{attribute 'global_init_slot' := '40510'}
VAR_GLOBAL
  TxTPlant_Facade_sObjectName                                            :T_BA_StateText:='FAS';
  TxTPlant_Facade_sDescription                                            :T_BA_StateText:='Fassade';
  TxTPlant_Natural_smoke_extraction_sObjectName                          :T_BA_StateText:='NRA';
  TxTPlant_Natural_smoke_extraction_sDescription                          :T_BA_StateText:='Natürlicher Rauchabzug';
  TxTPlant_Doors_gates_sluices_sObjectName                               :T_BA_StateText:='TUE';
  TxTPlant_Doors_gates_sluices_sDescription                               :T_BA_StateText:='Türen, Tore, Schleusen';
  TxTPlant_Smoke_and_heat_extraction_system_sObjectName                  :T_BA_StateText:='RWA';
  TxTPlant_Smoke_and_heat_extraction_system_sDescription                  :T_BA_StateText:='Rauch- und Wärmeabzugsanlage';
  TxTPlant_Sunlight_protection_sObjectName                               :T_BA_StateText:='SON';
  TxTPlant_Sunlight_protection_sDescription                               :T_BA_StateText:='Sonnenschutzanlage';
// 411 Abwasseranlagen
  TxTPlant_Separator_facility_sObjectName                                :T_BA_StateText:='ABS';
  TxTPlant_Separator_facility_sDescription                                :T_BA_StateText:='Abscheideranlage';
  TxTPlant_Lifting_system_sObjectName                                    :T_BA_StateText:='HBA';
  TxTPlant_Lifting_system_sDescription                                    :T_BA_StateText:='Hebeanlage';
  TxTPlant_Neutralisation_plant_sObjectName                              :T_BA_StateText:='NEU';
  TxTPlant_Neutralisation_plant_sDescription                              :T_BA_StateText:='Neutralisationsanlage';
// 412 Wasseranlagen
  TxTPlant_Trace_heating_sObjectName                                     :T_BA_StateText:='BGH';
  TxTPlant_Trace_heating_sDescription                                     :T_BA_StateText:='Begleitheizung';
  TxTPlant_Process_water_sObjectName                                     :T_BA_StateText:='BTW';
  TxTPlant_Process_water_sDescription                                     :T_BA_StateText:='Betriebswasser';
  TxTPlant_Well_water_sObjectName                                        :T_BA_StateText:='BWA';
  TxTPlant_Well_water_sDescription                                        :T_BA_StateText:='Brunnenwasser';
  TxTPlant_Dispensing_installation_sObjectName                           :T_BA_StateText:='DOS';
  TxTPlant_Dispensing_installation_sDescription                           :T_BA_StateText:='Dosieranlage';
  TxTPlant_Pressure_booster_system_sObjectName                           :T_BA_StateText:='DEA';
  TxTPlant_Pressure_booster_system_sDescription                           :T_BA_StateText:='Druckerhöhungsanlage';
  TxTPlant_Softening_unit_sObjectName                                    :T_BA_StateText:='EHA';
  TxTPlant_Softening_unit_sDescription                                    :T_BA_StateText:='Enthärtungsanlage';
// Trinkwasser
  TxTPlant_Drinking_water_heating_system_sObjectName                     :T_BA_StateText:='TWE';
  TxTPlant_Drinking_water_heating_system_sDescription                     :T_BA_StateText:='Trinkwassererwärmungsanlage';
  TxTPlant_Reverse_osmosis_system_sObjectName                            :T_BA_StateText:='UKO';
  TxTPlant_Reverse_osmosis_system_sDescription                            :T_BA_StateText:='Umkehrosmoseanlage';
  TxTPlant_Desalination_plant_sObjectName                                :T_BA_StateText:='VEA';
  TxTPlant_Desalination_plant_sDescription                                :T_BA_StateText:='Vollentsalzungsanlage';
// 421 Wärmeerzeugungsanlagen
  TxTPlant_BHKW_sObjectName                                              :T_BA_StateText:='BHK';
  TxTPlant_BHKW_sDescription                                              :T_BA_StateText:='BHKW';
  TxTPlant_Electric_heating_sObjectName                                  :T_BA_StateText:='EHZ';
  TxTPlant_Electric_heating_sDescription                                  :T_BA_StateText:='Elektroheizung';
  TxTPlant_District_heating_transfer_sObjectName                         :T_BA_StateText:='FWÜ';
  TxTPlant_District_heating_transfer_sDescription                         :T_BA_StateText:='Fernwärmeübergabe';
// Geothermieanlage
  TxTPlant_Boiler_sObjectName                                            :T_BA_StateText:='KES';
  TxTPlant_Boiler_sDescription                                            :T_BA_StateText:='Kessel';
  TxTPlant_Clean_steam_generation_sObjectName                            :T_BA_StateText:='RDE';
  TxTPlant_Clean_steam_generation_sDescription                            :T_BA_StateText:='Reindampferzeugung';
  TxTPlant_Solar_power_system_sObjectName                                :T_BA_StateText:='SOL';
  TxTPlant_Solar_power_system_sDescription                                :T_BA_StateText:='Solaranlage';
  TxTPlant_Heating_pump_sObjectName                                      :T_BA_StateText:='WPU';
  TxTPlant_Heating_pump_sDescription                                      :T_BA_StateText:='Wärmepumpe';
// 422 Wärmeverteilnetze
  TxTPlant_Pressure_maintenance_sObjectName                              :T_BA_StateText:='DHG';
  TxTPlant_Pressure_maintenance_sDescription                              :T_BA_StateText:='Druckhaltung';
  TxTPlant_Heating_circuit_sObjectName                                   :T_BA_StateText:='HZK';
  TxTPlant_Heating_circuit_sDescription                                   :T_BA_StateText:='Heizkreis';
  TxTPlant_Heating_sObjectName                                           :T_BA_StateText:='HZG';
  TxTPlant_Heating_sDescription                                           :T_BA_StateText:='Heizung';
  TxTPlant_Back_feed_system_sObjectName                                  :T_BA_StateText:='NSA';
  TxTPlant_Back_feed_system_sDescription                                  :T_BA_StateText:='Nachspeiseanlage';
  TxTPlant_Buffer_sObjectName                                            :T_BA_StateText:='PFS';
  TxTPlant_Buffer_sDescription                                            :T_BA_StateText:='Pufferspeicher';
  TxTPlant_Heat_distribution_network_sObjectName                         :T_BA_StateText:='WVN';
  TxTPlant_Heat_distribution_network_sDescription                         :T_BA_StateText:='Wärmeverteilnetz';
  TxTPlant_Heat_exchanger_sObjectName                                    :T_BA_StateText:='WTR';
  TxTPlant_Heat_exchanger_sDescription                                    :T_BA_StateText:='Wärmeüberträger';
// 423 Raumheizflächen
  TxTPlant_Concrete_core_activation_sObjectName                          :T_BA_StateText:='BKA';
  TxTPlant_Concrete_core_activation_sDescription                          :T_BA_StateText:='Betonkernaktivierung';
  TxTPlant_Overhead_heating_sObjectName                                  :T_BA_StateText:='DHZ';
  TxTPlant_Overhead_heating_sDescription                                  :T_BA_StateText:='Deckenheizung';
  TxTPlant_Ceiling_radiator_panels_sObjectName                           :T_BA_StateText:='DSP';
  TxTPlant_Ceiling_radiator_panels_sDescription                           :T_BA_StateText:='Deckenstrahlplatten';
  TxTPlant_Facade_heating_sObjectName                                    :T_BA_StateText:='FAH';
  TxTPlant_Facade_heating_sDescription                                    :T_BA_StateText:='Fassadenheizung';
  TxTPlant_Panel_heating_sObjectName                                     :T_BA_StateText:='FLH';
  TxTPlant_Panel_heating_sDescription                                     :T_BA_StateText:='Flächenheizung';
  TxTPlant_Underfloor_heating_sObjectName                                :T_BA_StateText:='FBH';
  TxTPlant_Underfloor_heating_sDescription                                :T_BA_StateText:='Fußbodenheizung';
  TxTPlant_Heated_chilled_ceiling_sObjectName                            :T_BA_StateText:='HKD';
  TxTPlant_Heated_chilled_ceiling_sDescription                            :T_BA_StateText:='Heiz-/Kühldecke';
  TxTPlant_Static_heating_sObjectName                                    :T_BA_StateText:='STH';
  TxTPlant_Static_heating_sDescription                                    :T_BA_StateText:='Statische Heizung';
// 430 Lufttechnische Anlagen
  TxTPlant_Extract_air_system_sObjectName                                :T_BA_StateText:='ABA';
  TxTPlant_Extract_air_system_sDescription                                :T_BA_StateText:='Abluftanlage';
  TxTPlant_Roof_air_heater_sObjectName                                   :T_BA_StateText:='DLH';
  TxTPlant_Roof_air_heater_sDescription                                   :T_BA_StateText:='Deckenlufterhitzer';
  TxTPlant_Circulatory_system_sObjectName                                :T_BA_StateText:='KVS';
  TxTPlant_Circulatory_system_sDescription                                :T_BA_StateText:='Kreislaufverbundsystem';
  TxTPlant_Air_processing_unit_sObjectName                               :T_BA_StateText:='LAZ';
  TxTPlant_Air_processing_unit_sDescription                               :T_BA_StateText:='Luftaufbereitungszentrale';
  TxTPlant_Mechanical_smoke_extraction_system_sObjectName                :T_BA_StateText:='MRA';
  TxTPlant_Mechanical_smoke_extraction_system_sDescription                :T_BA_StateText:='Maschinelle Rauchabzugsanlage';
  TxTPlant_Smoke_pressure_system_sObjectName                             :T_BA_StateText:='RDA';
  TxTPlant_Smoke_pressure_system_sDescription                             :T_BA_StateText:='Rauchdruckanlage';
  TxTPlant_Air_handling_unit_sObjectName                                 :T_BA_StateText:='RLT';
  TxTPlant_Air_handling_unit_sDescription                                 :T_BA_StateText:='Raumlufttechnik';
  TxTPlant_Partial_air_conditioning_system_sObjectName                   :T_BA_StateText:='TKA';
  TxTPlant_Partial_air_conditioning_system_sDescription                   :T_BA_StateText:='Teilklimaanlage';
  TxTPlant_Air_curtain_system_sObjectName                                :T_BA_StateText:='TLS';
  TxTPlant_Air_curtain_system_sDescription                                :T_BA_StateText:='Türluftschleieranlage';
  TxTPlant_Recirculating_air_system_sObjectName                          :T_BA_StateText:='ULA';
  TxTPlant_Recirculating_air_system_sDescription                          :T_BA_StateText:='Umluftanlage';
  TxTPlant_Full_air_conditioning_system_sObjectName                      :T_BA_StateText:='VKA';
  TxTPlant_Full_air_conditioning_system_sDescription                      :T_BA_StateText:='Vollklimaanlage';
  TxTPlant_Heat_recovery_system_sObjectName                              :T_BA_StateText:='WRG';
  TxTPlant_Heat_recovery_system_sDescription                              :T_BA_StateText:='Wärmerückgewinnungssystem';
  TxTPlant_Intake_air_system_sObjectName                                 :T_BA_StateText:='ZUA';
  TxTPlant_Intake_air_system_sDescription                                 :T_BA_StateText:='Zuluftanlage';
  TxTPlant_Smoke_extraction_system_sObjectName                           :T_BA_StateText:='ERA';
  TxTPlant_Smoke_extraction_system_sDescription                           :T_BA_StateText:='Entrauchungsanlage';
// 434 Kälteanlagen
  TxTPlant_Remote_cooling_transfer_sObjectName                           :T_BA_StateText:='FKÜ';
  TxTPlant_Remote_cooling_transfer_sDescription                           :T_BA_StateText:='Fernkälteübergabe';
  TxTPlant_Cooling_sObjectName                                           :T_BA_StateText:='KAE';
  TxTPlant_Cooling_sDescription                                           :T_BA_StateText:='Kälte';
  TxTPlant_Cooling_circuit_sObjectName                                   :T_BA_StateText:='KKR';
  TxTPlant_Cooling_circuit_sDescription                                   :T_BA_StateText:='Kältekreis';
  TxTPlant_Cooling_distribution_network_sObjectName                      :T_BA_StateText:='KVN';
  TxTPlant_Cooling_distribution_network_sDescription                      :T_BA_StateText:='Kälteverteilnetz';
  TxTPlant_Cold_water_generation_sObjectName                             :T_BA_StateText:='KWE';
  TxTPlant_Cold_water_generation_sDescription                             :T_BA_StateText:='Kaltwassererzeugung';
  TxTPlant_Electrical_cabinet_cooling_sObjectName                        :T_BA_StateText:='KVE';
  TxTPlant_Electrical_cabinet_cooling_sDescription                        :T_BA_StateText:='Kühlung Schaltschrank ';
  TxTPlant_Cooling_storage_sObjectName                                   :T_BA_StateText:='KSP';
  TxTPlant_Cooling_storage_sDescription                                   :T_BA_StateText:='Kältespeicher';
  TxTPlant_Chilled_ceiling_sObjectName                                   :T_BA_StateText:='KÜD';
  TxTPlant_Chilled_ceiling_sDescription                                   :T_BA_StateText:='Kühldecke';
  TxTPlant_Re_cooling_plant_sObjectName                                  :T_BA_StateText:='RKW';
  TxTPlant_Re_cooling_plant_sDescription                                  :T_BA_StateText:='Rückkühlwerk';
// 441 Hoch- und Mittelspannungsanlagen
  TxTPlant_Switchgear_sObjectName                                        :T_BA_StateText:='STA';
  TxTPlant_Switchgear_sDescription                                        :T_BA_StateText:='Schaltanlagen';
  TxTPlant_Transformer_sObjectName                                       :T_BA_StateText:='TRF';
  TxTPlant_Transformer_sDescription                                       :T_BA_StateText:='Transformator';
  TxTPlant_Medium_voltage_system_sObjectName                             :T_BA_StateText:='MSA';
  TxTPlant_Medium_voltage_system_sDescription                             :T_BA_StateText:='Mittelspannungsanlage';
  TxTPlant_Compensation_system_sObjectName                               :T_BA_StateText:='KOA';
  TxTPlant_Compensation_system_sDescription                               :T_BA_StateText:='Kompensationsanlage';
  TxTPlant_Frequency_converter_system_sObjectName                        :T_BA_StateText:='FUA';
  TxTPlant_Frequency_converter_system_sDescription                        :T_BA_StateText:='Frequenzumformeranlage';
// 442 Eigenstromversorgungsanlagen
  TxTPlant_Emissions_system_sObjectName                                  :T_BA_StateText:='AGA';
  TxTPlant_Emissions_system_sDescription                                  :T_BA_StateText:='Abgasanlage';
  TxTPlant_Battery_unit_sObjectName                                      :T_BA_StateText:='BAT';
  TxTPlant_Battery_unit_sDescription                                      :T_BA_StateText:='Batterieanlage';
  TxTPlant_Co_generation_unit_sObjectName                                :T_BA_StateText:='BHK';
  TxTPlant_Co_generation_unit_sDescription                                :T_BA_StateText:='Blockheizkraftwerk';
  TxTPlant_Fuel_supply_sObjectName                                       :T_BA_StateText:='BRV';
  TxTPlant_Fuel_supply_sDescription                                       :T_BA_StateText:='Brennstoffversorgung';
  TxTPlant_Standby_power_system_sObjectName                              :T_BA_StateText:='ESA';
  TxTPlant_Standby_power_system_sDescription                              :T_BA_StateText:='Ersatzstromanlage';
  TxTPlant_Photovoltaic_system_sObjectName                               :T_BA_StateText:='PVA';
  TxTPlant_Photovoltaic_system_sDescription                               :T_BA_StateText:='Fotovoltaikanlage';
  TxTPlant_Uninterruptible_power_supply_sObjectName                      :T_BA_StateText:='USV';
  TxTPlant_Uninterruptible_power_supply_sDescription                      :T_BA_StateText:='Unterbrechungsfreie Stromversorgung';
// 443 Niederspannungsschaltanlagen
  TxTPlant_General_power_supply_sObjectName                              :T_BA_StateText:='ASV';
  TxTPlant_General_power_supply_sDescription                              :T_BA_StateText:='Allgemeine Stromversorgung';
  TxTPlant_Safety_power_supply_sObjectName                               :T_BA_StateText:='SSV';
  TxTPlant_Safety_power_supply_sDescription                               :T_BA_StateText:='Sicherheitsstromversorgung';
  TxTPlant_Lighting_sObjectName                                          :T_BA_StateText:='BEL';
  TxTPlant_Lighting_sDescription                                          :T_BA_StateText:='Beleuchtungsanlage';
  TxTPlant_Emergency_lighting_sObjectName                                :T_BA_StateText:='SIB';
  TxTPlant_Emergency_lighting_sDescription                                :T_BA_StateText:='Sicherheitsbeleuchtung';
// 451 Telekommunikationsanlagen
  TxTPlant_Telecommunications_system_sObjectName                         :T_BA_StateText:='TEL';
  TxTPlant_Telecommunications_system_sDescription                         :T_BA_StateText:='Telekommunikationsanlage';
// 452 Such- und Signalanlagen
  TxTPlant_Call_signalling_system_sObjectName                            :T_BA_StateText:='LRA';
  TxTPlant_Call_signalling_system_sDescription                            :T_BA_StateText:='Lichtrufanlage';
  TxTPlant_Door_intercom_and_door_opener_system_sObjectName              :T_BA_StateText:='TÜA';
  TxTPlant_Door_intercom_and_door_opener_system_sDescription              :T_BA_StateText:='Türsprech- und -öffneranlage';
  TxTPlant_Paging_system_sObjectName                                     :T_BA_StateText:='PRA';
  TxTPlant_Paging_system_sDescription                                     :T_BA_StateText:='Personenrufanlage';
// 453 Zeitdienstanlagen
  TxTPlant_Clock_and_time_recording_system_sObjectName                   :T_BA_StateText:='ZEA';
  TxTPlant_Clock_and_time_recording_system_sDescription                   :T_BA_StateText:='Uhren- und Zeiterfassungsanlage';
// 454 Elektroakustische Anlagen
  TxTPlant_Electro_acoustic_sound_systems_sObjectName                    :T_BA_StateText:='ELA';
  TxTPlant_Electro_acoustic_sound_systems_sDescription                    :T_BA_StateText:='Elektroakustische Anl. , Beschallung';
  TxTPlant_Conference_and_interpreting_equipment_sObjectName             :T_BA_StateText:='KDA';
  TxTPlant_Conference_and_interpreting_equipment_sDescription             :T_BA_StateText:='Konferenz- und Dolmetscheranlage';
  TxTPlant_Intercom_system_sObjectName                                   :T_BA_StateText:='GSA';
  TxTPlant_Intercom_system_sDescription                                   :T_BA_StateText:='Gegensprechanlage';
  TxTPlant_Voice_alarm_system_sObjectName                                :T_BA_StateText:='SAA';
  TxTPlant_Voice_alarm_system_sDescription                                :T_BA_StateText:='Sprachalarmierungsanlage';
  TxTPlant_Intercommunication_systems_sObjectName                        :T_BA_StateText:='WSA';
  TxTPlant_Intercommunication_systems_sDescription                        :T_BA_StateText:='Wechselsprechanlagen';
// 455 Fernseh- und Antennenanlagen
  TxTPlant_Television_system_sObjectName                                 :T_BA_StateText:='TVA';
  TxTPlant_Television_system_sDescription                                 :T_BA_StateText:='Fernsehanlage';
  TxTPlant_Transmitting_and_receiving_antenna_system_sObjectName         :T_BA_StateText:='SEA';
  TxTPlant_Transmitting_and_receiving_antenna_system_sDescription         :T_BA_StateText:='Sende- und Empfangsantennenanlage';
  TxTPlant_BOS_radio_system_sObjectName                                  :T_BA_StateText:='BOS';
  TxTPlant_BOS_radio_system_sDescription                                  :T_BA_StateText:='BOS-Funkanlage';
// 456 Gefahrenmelde- und Alarmanlagen
  TxTPlant_Fire_detection_and_alarm_system_sObjectName                   :T_BA_StateText:='BMA';
  TxTPlant_Fire_detection_and_alarm_system_sDescription                   :T_BA_StateText:='Brandmeldeanlage';
  TxTPlant_Carbon_monoxide_warning_system_sObjectName                    :T_BA_StateText:='COW';
  TxTPlant_Carbon_monoxide_warning_system_sDescription                    :T_BA_StateText:='CO-Warnanlage';
  TxTPlant_Burglar_alarm_system_sObjectName                              :T_BA_StateText:='EMA';
  TxTPlant_Burglar_alarm_system_sDescription                              :T_BA_StateText:='Einbruchmeldeanlage';
  TxTPlant_Fire_control_panel_sObjectName                                :T_BA_StateText:='FWT';
  TxTPlant_Fire_control_panel_sDescription                                :T_BA_StateText:='Feuerwehrtableau';
  TxTPlant_Escape_route_protection_system_sObjectName                    :T_BA_StateText:='FWS';
  TxTPlant_Escape_route_protection_system_sDescription                    :T_BA_StateText:='Fluchtwegsicherungsanlage';
  TxTPlant_Hazard_detection_system_sObjectName                           :T_BA_StateText:='GMA';
  TxTPlant_Hazard_detection_system_sDescription                           :T_BA_StateText:='Gefahrenmeldeanlage';
  TxTPlant_Gas_warning_system_sObjectName                                :T_BA_StateText:='GWA';
  TxTPlant_Gas_warning_system_sDescription                                :T_BA_StateText:='Gaswarnanlage';
  TxTPlant_Smoke_aspiration_system_sObjectName                           :T_BA_StateText:='RAS';
  TxTPlant_Smoke_aspiration_system_sDescription                           :T_BA_StateText:='Rauchansaugsystem';
  TxTPlant_Room_observation_system_sObjectName                           :T_BA_StateText:='RBA';
  TxTPlant_Room_observation_system_sDescription                           :T_BA_StateText:='Raumbeobachtungsanlage';
  TxTPlant_Robbery_alarm_system_sObjectName                              :T_BA_StateText:='ÜFA';
  TxTPlant_Robbery_alarm_system_sDescription                              :T_BA_StateText:='Überfallmeldeanlage';
  TxTPlant_Guard_control_system_sObjectName                              :T_BA_StateText:='WKA';
  TxTPlant_Guard_control_system_sDescription                              :T_BA_StateText:='Wächterkontrollanlage';
  TxTPlant_Emergency_call_system_sObjectName                             :T_BA_StateText:='NOT';
  TxTPlant_Emergency_call_system_sDescription                             :T_BA_StateText:='Notrufanlage';
  TxTPlant_Access_control_system_sObjectName                             :T_BA_StateText:='ZKS';
  TxTPlant_Access_control_system_sDescription                             :T_BA_StateText:='Zugangskontrollsystem';
// 457 Übertragungsnetze
  TxTPlant_Networks_for_the_transmission_voice_text_etc_sObjectName      :T_BA_StateText:='LAN';
  TxTPlant_Networks_for_the_transmission_voice_text_etc_sDescription      :T_BA_StateText:='Netzw.  Daten, Sprache, Text etc';
// 459 Fernmelde- und informationstechnische Anlagen, Sonstiges
  TxTPlant_Remote_control_systems_sObjectName                            :T_BA_StateText:='FWA';
  TxTPlant_Remote_control_systems_sDescription                            :T_BA_StateText:='Fernwirkanlagen';
  TxTPlant_Parking_guidance_systems_sObjectName                          :T_BA_StateText:='PLS';
  TxTPlant_Parking_guidance_systems_sDescription                          :T_BA_StateText:='Parkleitsysteme';
// 460 Förderanlagen
  TxTPlant_File_transportation_systems_sObjectName                       :T_BA_StateText:='ATA';
  TxTPlant_File_transportation_systems_sDescription                       :T_BA_StateText:='Aktentransportanlagen';
  TxTPlant_Lift_sObjectName                                              :T_BA_StateText:='AUF';
  TxTPlant_Lift_sDescription                                              :T_BA_StateText:='Aufzug';
  TxTPlant_Inspection_systems_sObjectName                                :T_BA_StateText:='BFA';
  TxTPlant_Inspection_systems_sDescription                                :T_BA_StateText:='Befahranlagen';
  TxTPlant_Moving_walkways_sObjectName                                   :T_BA_StateText:='FST';
  TxTPlant_Moving_walkways_sDescription                                   :T_BA_StateText:='Fahrsteige';
  TxTPlant_Escalators_sObjectName                                        :T_BA_StateText:='FTR';
  TxTPlant_Escalators_sDescription                                        :T_BA_StateText:='Fahrtreppen';
  TxTPlant_External_lifts_sObjectName                                    :T_BA_StateText:='FSA';
  TxTPlant_External_lifts_sDescription                                    :T_BA_StateText:='Fassadenaufzüge';
  TxTPlant_Baggage_conveyor_system_sObjectName                           :T_BA_StateText:='GFA';
  TxTPlant_Baggage_conveyor_system_sDescription                           :T_BA_StateText:='Gepäckförderanlage';
  TxTPlant_Pneumatic_delivery_systems_sObjectName                        :T_BA_StateText:='RPA';
  TxTPlant_Pneumatic_delivery_systems_sDescription                        :T_BA_StateText:='Rohrpostanlagen';
  TxTPlant_Goods_transportation_facilities_sObjectName                   :T_BA_StateText:='WTA';
  TxTPlant_Goods_transportation_facilities_sDescription                   :T_BA_StateText:='Warentransportanlagen';
// 470 Nutzerspezifische Anlagen
// 471 Küchentechnische Anlagen
  TxTPlant_Small_refrigeration_unit_sObjectName                          :T_BA_StateText:='KLK';
  TxTPlant_Small_refrigeration_unit_sDescription                          :T_BA_StateText:='Kleinkälteanlage';
// 472 Wäscherei- und Reinigungsanlagen
  TxTPlant_Disinfection_unit_sObjectName                                 :T_BA_StateText:='DES';
  TxTPlant_Disinfection_unit_sDescription                                 :T_BA_StateText:='Desinfektionsanlage';
  TxTPlant_Cleaning_unit_sObjectName                                     :T_BA_StateText:='REA';
  TxTPlant_Cleaning_unit_sDescription                                     :T_BA_StateText:='Reinigungsanlage';
  TxTPlant_Sterilisation_systems_sObjectName                             :T_BA_StateText:='STR';
  TxTPlant_Sterilisation_systems_sDescription                             :T_BA_StateText:='Sterilisationseinrichtungen';
  TxTPlant_Water_treatment_system_sObjectName                            :T_BA_StateText:='WAA';
  TxTPlant_Water_treatment_system_sDescription                            :T_BA_StateText:='Wasseraufbereitungsanlage';
  TxTPlant_Laundry_system_sObjectName                                    :T_BA_StateText:='WÄA';
  TxTPlant_Laundry_system_sDescription                                    :T_BA_StateText:='Wäschereianlage';
// 473 Medienversorgungsanlagen
  TxTPlant_Compressed_air_supply_system_sObjectName                      :T_BA_StateText:='DRL';
  TxTPlant_Compressed_air_supply_system_sDescription                      :T_BA_StateText:='Druckluftversorgungsanlage';
  TxTPlant_Pressure_regulator_unit_sObjectName                           :T_BA_StateText:='DRA';
  TxTPlant_Pressure_regulator_unit_sDescription                           :T_BA_StateText:='Druckregelanlage';
  TxTPlant_Media_supply_system_sObjectName                               :T_BA_StateText:='MVA';
  TxTPlant_Media_supply_system_sDescription                               :T_BA_StateText:='Medienversorgungsanlage';
  TxTPlant_Medical_and_technical_gases_sObjectName                       :T_BA_StateText:='MTG';
  TxTPlant_Medical_and_technical_gases_sDescription                       :T_BA_StateText:='Medizinische und technische Gase';
  TxTPlant_Vacuum_unit_sObjectName                                       :T_BA_StateText:='VAK';
  TxTPlant_Vacuum_unit_sDescription                                       :T_BA_StateText:='Vakuumanlage';
// 474 Medizin- und labortechnische Anlagen
  TxTPlant_Medical_technical_plant_sObjectName                           :T_BA_StateText:='MED';
  TxTPlant_Medical_technical_plant_sDescription                           :T_BA_StateText:='Medizintechnische Anlagen';
  TxTPlant_Medical_gas_supply_sObjectName                                :T_BA_StateText:='MGV';
  TxTPlant_Medical_gas_supply_sDescription                                :T_BA_StateText:='Medizinische Gasversorgung';
  TxTPlant_Laboratory_equipment_sObjectName                              :T_BA_StateText:='LAB';
  TxTPlant_Laboratory_equipment_sDescription                              :T_BA_StateText:='Labortechnische Anlagen (allgemein)';
// 475 Feuerlöschanlagen
  TxTPlant_Fire_extinguisher_sObjectName                                 :T_BA_StateText:='FLA';
  TxTPlant_Fire_extinguisher_sDescription                                 :T_BA_StateText:='Feuerlöschanlage';
  TxTPlant_Gas_extinguishing_system_sObjectName                          :T_BA_StateText:='GLA';
  TxTPlant_Gas_extinguishing_system_sDescription                          :T_BA_StateText:='Gaslöschanlage';
  TxTPlant_Fire_extinguishing_system_sObjectName                         :T_BA_StateText:='LÖS';
  TxTPlant_Fire_extinguishing_system_sDescription                         :T_BA_StateText:='Löschanlage (allgemein)';
  TxTPlant_Mist_extinguishing_system_sObjectName                         :T_BA_StateText:='NLA';
  TxTPlant_Mist_extinguishing_system_sDescription                         :T_BA_StateText:='Nebellöschanlage';
  TxTPlant_NOX_system_sObjectName                                        :T_BA_StateText:='NOX';
  TxTPlant_NOX_system_sDescription                                        :T_BA_StateText:='NOX-Anlage';
  TxTPlant_Sprinkler_system_sObjectName                                  :T_BA_StateText:='SPR';
  TxTPlant_Sprinkler_system_sDescription                                  :T_BA_StateText:='Sprinkleranlage';
  TxTPlant_Wall_hydrant_system_sObjectName                               :T_BA_StateText:='WHA';
  TxTPlant_Wall_hydrant_system_sDescription                               :T_BA_StateText:='Wandhydrantenanlage';
// 478 Entsorgungsanlagen
  TxTPlant_Waste_disposal_system_sObjectName                             :T_BA_StateText:='AEA';
  TxTPlant_Waste_disposal_system_sDescription                             :T_BA_StateText:='Abfallentsorgungsanlage';
  TxTPlant_Media_disposal_system_sObjectName                             :T_BA_StateText:='MEA';
  TxTPlant_Media_disposal_system_sDescription                             :T_BA_StateText:='Medienentsorgungsanlage';
  TxTPlant_Vacuum_cleaning_systems_sObjectName                           :T_BA_StateText:='SSA';
  TxTPlant_Vacuum_cleaning_systems_sDescription                           :T_BA_StateText:='Staubsauganlagen';
// 480 Gebäudeautomation
  TxTPlant_Information_focal_point_sObjectName                           :T_BA_StateText:='ISP';
  TxTPlant_Information_focal_point_sDescription                           :T_BA_StateText:='Informationsschwerpunkt';
  TxTPlant_Weather_station_sObjectName                                   :T_BA_StateText:='WET';
  TxTPlant_Weather_station_sDescription                                   :T_BA_StateText:='Wetterstation';
  TxTPlant_Management_and_operating_equipment_sObjectName                :T_BA_StateText:='MBE';
  TxTPlant_Management_and_operating_equipment_sDescription                :T_BA_StateText:='Management- und Bedieneinrichtungen';
  TxTPlant_Room_automation_sObjectName                                   :T_BA_StateText:='RAU';
  TxTPlant_Room_automation_sDescription                                   :T_BA_StateText:='Raumautomation';
  TxTPlant_Room_automation_system_distributor_sObjectName                :T_BA_StateText:='RAV';
  TxTPlant_Room_automation_system_distributor_sDescription                :T_BA_StateText:='Raumautomation-Systemverteiler';
  TxTPlant_Control_cabinet_sObjectName                                   :T_BA_StateText:='SSK';
  TxTPlant_Control_cabinet_sDescription                                   :T_BA_StateText:='Schaltschrank';
  TxTPlant_Settings_sObjectName                                          :T_BA_StateText:='ALP';
  TxTPlant_Settings_sDescription                                          :T_BA_StateText:='Anlagenparameter';
  TxTPlant_EventGroups_sObjectName                                       :T_BA_StateText:='ERG';
  TxTPlant_EventGroups_sDescription                                       :T_BA_StateText:='Meldeklassen';
  TxTPlant_Global_Building_Data_sObjectName                              :T_BA_StateText:='GGL';
  TxTPlant_Global_Building_Data_sDescription                              :T_BA_StateText:='globale Gebäudedaten';
// 540 Technische Anlagen in Außenanlagen
  TxTPlant_Rainwater_retention_basin_sObjectName                         :T_BA_StateText:='RRB';
  TxTPlant_Rainwater_retention_basin_sDescription                         :T_BA_StateText:='Regenrückhaltebecken';
  TxTPlant_Cistern_system_sObjectName                                    :T_BA_StateText:='ZTA';
  TxTPlant_Cistern_system_sDescription                                    :T_BA_StateText:='Zisternenanlage';
END_VAR

// ---- Templates/GVLs/Language/German/TxtTrade_DE.TcGVL
{region '#Template'}
	{attribute 'Version' := '1.2.0.0'}
	{attribute 'Tags' := '"LCID": "1031", "Text": "GVL, DPAD, Trades, ObjectName, Description"'}
	{attribute 'Tags' := '"LCID": "1033", "Text": "GVL, DPAD, Trades, ObjectName, Description"'}
	{attribute 'Description' := '"LCID": "1031", "Text": "Textliste Gewerke"'}
	{attribute 'Description' := '"LCID": "1033", "Text": "Text list trades"'}
{endregion}

{attribute 'global_init_slot' := '40510'}
VAR_GLOBAL
  TxtTrade_Doors_gates_windows_sun_protection_sObjectName                :T_BA_StateText:='TTF';
  TxtTrade_Doors_gates_windows_sun_protection_sDescription                :T_BA_StateText:='Türen, Tore, Fenster, Sonnenschutz';
  TxtTrade_Sewage_water_and_gas_plants_sObjectName                       :T_BA_StateText:='GWA';
  TxtTrade_Sewage_water_and_gas_plants_sDescription                       :T_BA_StateText:='Abwasser-, Wasser-, Gasanlagen';
  TxtTrade_Heat_supply_systems_sObjectName                               :T_BA_StateText:='HZG';
  TxtTrade_Heat_supply_systems_sDescription                               :T_BA_StateText:='Wärmeversorgungsanlagen';
  TxtTrade_Air_conditioning_sObjectName                                  :T_BA_StateText:='LTA';
  TxtTrade_Air_conditioning_sDescription                                  :T_BA_StateText:='Lufttechnische Anlagen';
  TxtTrade_Refrigeration_systems_sObjectName                             :T_BA_StateText:='KAE';
  TxtTrade_Refrigeration_systems_sDescription                             :T_BA_StateText:='Kälteanlagen';
  TxtTrade_High_voltage_systems_sObjectName                              :T_BA_StateText:='ELT';
  TxtTrade_High_voltage_systems_sDescription                              :T_BA_StateText:='Starkstromanlagen';
  TxtTrade_Telecommunication_and_information_technology_sObjectName      :T_BA_StateText:='FIA';
  TxtTrade_Telecommunication_and_information_technology_sDescription      :T_BA_StateText:='Fernm.- und informationstech. Anlagen';
  TxtTrade_Hazard_detection_and_alarm_systems_sObjectName                :T_BA_StateText:='GMA';
  TxtTrade_Hazard_detection_and_alarm_systems_sDescription                :T_BA_StateText:='Gefahrenmelde- und Alarmanlagen';
  TxtTrade_Conveyors_sObjectName                                         :T_BA_StateText:='FTA';
  TxtTrade_Conveyors_sDescription                                         :T_BA_StateText:='Förderanlagen';
  TxtTrade_Kitchen_technology_systems_sObjectName                        :T_BA_StateText:='KTA';
  TxtTrade_Kitchen_technology_systems_sDescription                        :T_BA_StateText:='Küchentechnische Anlagen';
  TxtTrade_Laundry_and_cleaning_systems_sObjectName                      :T_BA_StateText:='WAR';
  TxtTrade_Laundry_and_cleaning_systems_sDescription                      :T_BA_StateText:='Wäscherei- und Reinigungsanlagen';
  TxtTrade_Media_supply_systems_sObjectName                              :T_BA_StateText:='MVA';
  TxtTrade_Media_supply_systems_sDescription                              :T_BA_StateText:='Medienversorgungsanlagen';
  TxtTrade_Medical_and_laboratory_equipment_sObjectName                  :T_BA_StateText:='MED';
  TxtTrade_Medical_and_laboratory_equipment_sDescription                  :T_BA_StateText:='Medizin- und labortechnische Anlagen';
  TxtTrade_Fire_extinguishing_systems_sObjectName                        :T_BA_StateText:='FLA';
  TxtTrade_Fire_extinguishing_systems_sDescription                        :T_BA_StateText:='Feuerlöschanlagen';
  TxtTrade_Bathing_facilities_sObjectName                                :T_BA_StateText:='BTA';
  TxtTrade_Bathing_facilities_sDescription                                :T_BA_StateText:='Badetechnische Anlagen';
  TxtTrade_Process_heating_cooling_and_air_systems_sObjectName           :T_BA_StateText:='PRO';
  TxtTrade_Process_heating_cooling_and_air_systems_sDescription           :T_BA_StateText:='Prozesswärme-, -kälte- und -luftanlagen';
  TxtTrade_Waste_disposal_facilities_sObjectName                         :T_BA_StateText:='ENT';
  TxtTrade_Waste_disposal_facilities_sDescription                         :T_BA_StateText:='Entsorgungsanlagen';
  TxtTrade_Building_automation_and_control_systems_general_sObjectName   :T_BA_StateText:='GAS';
  TxtTrade_Building_automation_and_control_systems_general_sDescription   :T_BA_StateText:='Gebäudeautomation allgemein';
  TxtTrade_Automation_focal_point_information_focal_point_sObjectName    :T_BA_StateText:='ASP';
  TxtTrade_Automation_focal_point_information_focal_point_sDescription    :T_BA_StateText:='Automationsschwerpunkt';
  TxtTrade_Room_automation_sObjectName                                   :T_BA_StateText:='RAU';
  TxtTrade_Room_automation_sDescription                                   :T_BA_StateText:='Raumautomation';
  TxtTrade_Outdoor_devices_sObjectName                                   :T_BA_StateText:='AUG';
  TxtTrade_Outdoor_devices_sDescription                                   :T_BA_StateText:='Außengeräte';
END_VAR

// ---- Templates/GVLs/Site/Site.TcGVL
{region '#Template'}
	{attribute 'Version' := '1.0.0.0'}
	{attribute 'Tags' := '"LCID": "1031", "Text": "GVL, Publisher, Subscriber"'}
	{attribute 'Tags' := '"LCID": "1033", "Text": "GVL, Publisher, Subscriber"'}
	{attribute 'Description' := '"LCID": "1031", "Text": "Ams NetId, Subject"'}
	{attribute 'Description' := '"LCID": "1033", "Text": "Ams NetId, Subject"'}
{endregion}

{attribute 'qualified_only'}
VAR_GLOBAL	
	Self_NetId						: T_BA_MedString	:= '127.0.0.1.1.1';
	Ipc1_NetId						: T_BA_MedString	:= Self_NetId;
	Ipc2_NetId						: T_BA_MedString	:= Self_NetId;
	Ipc3_NetId						: T_BA_MedString	:= Self_NetId;
	Ipc4_NetId						: T_BA_MedString	:= Self_NetId;
	Ipc5_NetId						: T_BA_MedString	:= Self_NetId;
	                            	
	GeneralSettings_Subject			: T_BA_MedString	:= 'GeneralSettings';	
	GeneralSettings_NetId			: T_BA_MedString	:= Self_NetId;	
		                        	
	WeatherStation_Subject			: T_BA_MedString	:= 'WeatherStation';
	WeatherStation_NetId			: T_BA_MedString	:= Self_NetId;
                                	
	FacadeNorth_NetId				: T_BA_MedString	:= Ipc1_NetId;
	FacadeNorth_Subject				: T_BA_MedString	:= 'FcdNorth.FacadeSunBlind';
	FacadeEast_NetId				: T_BA_MedString	:= Ipc1_NetId;
	FacadeEast_Subject				: T_BA_MedString	:= 'FcdEast.FacadeSunBlind';
	FacadeSouth_NetId				: T_BA_MedString	:= Ipc1_NetId;
	FacadeSouth_Subject				: T_BA_MedString	:= 'FcdSouth.FacadeSunBlind';
	FacadeWest_NetId				: T_BA_MedString	:= Ipc1_NetId;
	FacadeWest_Subject				: T_BA_MedString	:= 'FcdWest.FacadeSunBlind';
                                	
	Building_NetId					: T_BA_MedString	:= Ipc1_NetId;
	BuildingAlarms_Subject			: T_BA_MedString	:= 'BuildingAlarms';
	BuildingMode_Subject			: T_BA_MedString	:= 'BuildingMode';
	BuildingEnergyLevel_Subject		: T_BA_MedString	:= 'BuildingEnergyLevel';
	BuildingSpRmT_Subject			: T_BA_MedString	:= 'BuildingSpRmT';
	BuildingSunProtection_Subject	: T_BA_MedString	:= 'BuildingSunProtection';
END_VAR

// ---- POUs/MAIN.TcPOU
PROGRAM MAIN
VAR
	DPAD		: FB_BA_CarelessDPAD := (
					aIdentifier := [
	(* Level 1 *)		(eMode:=E_BA_DPADMode.eInclude,		eNodeType:=E_BA_NodeType.eLocation,			sSeparator_ObjectName := '-', 	sSeparator_Description := ' - ',	nIndexDigits := 0),
	(* Level 2 *)		(eMode:=E_BA_DPADMode.eInclude,		eNodeType:=E_BA_NodeType.eBuilding,			sSeparator_ObjectName := '-', 	sSeparator_Description := ' - ',	nIndexDigits := 0),
	(* Level 3 *)		(eMode:=E_BA_DPADMode.eInclude,		eNodeType:=E_BA_NodeType.eControlCabinet,	sSeparator_ObjectName := '-', 	sSeparator_Description := ' - ',	nIndexDigits := 0),
	(* Level 4 *)		(eMode:=E_BA_DPADMode.eInclude,		eNodeType:=E_BA_NodeType.eFloor,			sSeparator_ObjectName := '-', 	sSeparator_Description := ' - ',	nIndexDigits := 0),
	(* Level 5 *)		(eMode:=E_BA_DPADMode.eInclude,		eNodeType:=E_BA_NodeType.eTrade,			sSeparator_ObjectName := '-', 	sSeparator_Description := ' - ',	nIndexDigits := 0),
	(* Level 6 *)		(eMode:=E_BA_DPADMode.eInclude,		eNodeType:=E_BA_NodeType.ePlant,			sSeparator_ObjectName := '-', 	sSeparator_Description := ' - ',	nIndexDigits := 0),
	(* Level 7 *)		(eMode:=E_BA_DPADMode.eInclude,		eNodeType:=E_BA_NodeType.eAggregate,		sSeparator_ObjectName := '-', 	sSeparator_Description := ' - ',	nIndexDigits := 2),
	(* Level 8 *)		(eMode:=E_BA_DPADMode.eInclude,		eNodeType:=E_BA_NodeType.eFunction,			sSeparator_ObjectName := '-', 	sSeparator_Description := ' - ',	nIndexDigits := 2)
					]
				);		
		 
//	Level 1 Standort bzw. Ort oder Stadt 
//	Level 1 Site respectively location or town
	SiteA		: FB_BA_View := (
					sObjectName		:= 'A',		
					sDescription	:= 'A',	
					eDPADMode		:= E_BA_DPADMode.eInclude				
				); 				
//	Level 2 Gebäude 	
//	Level 2 Building 	
		B			: FB_BA_View := (
						iParent 		:= SiteA,
						sObjectName		:= 'B',		
						sDescription	:= 'B',	
						eDPADMode		:= E_BA_DPADMode.eInclude					
					);     
// Level 3 ISP -> Informationsschwerpunkt
// Level 3 IFP -> information focal point 	 	                                                                                   	
			IFP			: FB_BA_View := (
							iParent 		:= B,
							sObjectName		:= 'I',		
							sDescription	:= 'IFP',	
							eDPADMode		:= E_BA_DPADMode.eInclude				
						);     
// Level 4 Stockwerk 	->	O01 = Obergeschoss 01, U01 = Untergeschoss 01,  E00 = Ergeschoss
// Level 4 floor ->	F01 = floor 01, B01 = basement 01,  GFL = Ground floor  						
				F01			: FB_BA_View := (
								iParent 		:= IFP,
								sObjectName		:= 'F01',		
								sDescription	:= 'Floor 01',
								eDPADMode		:= E_BA_DPADMode.eInclude					
							);     	
// Level 5 Gewerk Wärmeversorgungsanlagen  
// Level 5 Trade Heat supply systems, heat distribution  --> 	HD = heat distribution, HG = heat generation
					H			: FB_BA_H := (
									iParent 		:= F01,
									sObjectName		:= 'HTG',		
									sDescription	:= 'Heat supply systems',
									eDPADMode		:= E_BA_DPADMode.eInclude			
								);     	 	
// Level 5 Gewerk Gebäudeautomation Allgemein   
// Level 5 Trade General                                                                                       	
					G			: FB_BA_General := (
									iParent 		:= F01,
									sObjectName		:= 'BAG',
									sDescription	:= 'General',
									eDPADMode		:= E_BA_DPADMode.eInclude					
								);     	 											   	 											
// Level 5 Gewerk Luftechnische Anlagen      
// Level 5 Trade ventilation system                                                                                	
					AC			: FB_BA_AC := (
									iParent 		:= F01,
									sObjectName		:= 'AC_',
									sDescription	:= 'Air conditioning',
									eDPADMode		:= E_BA_DPADMode.eInclude
								);     	
// Level 5 Gewerk Raumautomation    
// Level 5 Trade room automation                                                                              	

								
// Level 5 Gewerk Außengeräte   
// Level 5 Trade Outdoor devices     
					OD			: FB_BA_OD := (
									iParent			:= F01,
									sObjectName		:= 'ODD',
									sDescription	:= 'Outdoor devices',
									eDPADMode		:= E_BA_DPADMode.eInclude
								);
END_VAR

//	Level 1 Standort bzw. Ort oder Stadt 	Site respectively location or town
SiteA();
//	Level 2 Gebäude 	Building		
	B();
// Level 3 ISP -> Informationsschwerpunkt	information focal point 
		IFP();
// Level 4 Stockwerk -->	O01 = Obergeschoss 01, U01 = Untergeschoss 01,  E00 = Ergeschoss 	floor ->	F01 = floor 01, B01 = basement 01,  GFL = Ground floor
			F01();
// Level 5 Gewerk Wärmeversorgungsanlagen	Heat supply systems	
				H(); 								
// Level 5 Gewerk Allgemein		Trade General			
				G(); 								
// Level 5 Gewerk Luftechnische Anlagen		Trade ventilation system	
				AC(); 								
// Level 5 Gewerk Raumautomation	Trade room automation 

// Level 5 Gewerk Außengeräte 	Trade Outdoor devices
				OD();

END_PROGRAM

// ---- Templates/POUs/Trade/HeatingSystem/FB_BA_H.TcPOU
{region '#Template'}
	{attribute 'Version' := '1.2.1.0'}
	{attribute 'Tags' := '"LCID": "1031", "Text": "Trade, Plant, Heating System"'}
	{attribute 'Tags' := '"LCID": "1033", "Text": "Trade, Plant, Heating System"'}
	{attribute 'Using' := '"Type": "Template", "URI": "Site"'}
	{attribute 'Description' := '"LCID": "1031", "Text": "Aufruf der Anlagen des Gewerks Heizsysteme"'}
	{attribute 'Description' := '"LCID": "1033", "Text": "Calling the plants of the trade heating system"'}
{endregion}
FUNCTION_BLOCK FB_BA_H EXTENDS FB_BA_View
VAR_INPUT CONSTANT
	HTC01				: FB_BA_H_HtgCir01;		
END_VAR
VAR_INPUT
END_VAR
VAR_OUTPUT
END_VAR
VAR
END_VAR

SUPER^(); // FB_BA_View
HTC01(); // FB_BA_H_HtgCir01

METHOD FB_init : BOOL
VAR_INPUT
	bInitRetains : BOOL; // if TRUE, the retain variables are initialized (warm start / cold start)
	bInCopyCode : BOOL;  // if TRUE, the instance afterwards gets moved into the copy code (online change)
END_VAR
HTC01.iParent 				:= THIS^;	
HTC01.sObjectName				:= '{HTC01}';							
HTC01.sDescription			:= '{Heating circuit}';	
HTC01.eDPADMode				:= E_BA_DPADMode.eInclude;

HTC01.GeneralSettings.Subject	:= Site.GeneralSettings_Subject;
HTC01.GeneralSettings.sTarget	:= Site.GeneralSettings_NetId;
END_METHOD

END_FUNCTION_BLOCK

// ---- Templates/POUs/Trade/HeatingSystem/Distribution/HeatingCircuit/FB_BA_H_HtgCir01.TcPOU
{region '#Template'}
	{attribute 'Version' := '1.2.1.0'}
	{attribute 'Tags' := '"LCID": "1031", "Text": "H, Plant, HtgCir, Heating circuit"'}
	{attribute 'Tags' := '"LCID": "1033", "Text": "H, Plant, HtgCir, Heating circuit"'}
	{attribute 'Using' := '"Type": "Template", "URI": "Site"'}
	{attribute 'Description' := '"LCID": "1031", "Text": "Heizkreis"'}
	{attribute 'Description' := '"LCID": "1033", "Text": "Heating circuit"'}
{endregion}
FUNCTION_BLOCK FB_BA_H_HtgCir01 EXTENDS FB_BA_View
VAR_INPUT
END_VAR
VAR_OUTPUT
	eOpMod 					: E_BA_EnergyLvl;
	bRls					: BOOL;	
	fSp    					: REAL;
	bPu    					: BOOL;
	fVlv   					: REAL;
END_VAR
VAR_INPUT CONSTANT
	TFl						: FB_BA_SensorAnalog_IO;												
	TRt						: FB_BA_SensorAnalog_IO;																									
	Vlv						: FB_BA_Vlv;									
	Pu						: FB_BA_Pu1st;	
	Sp						: FB_BA_H_HtgCir_Sp;												
	OpMod					: FB_BA_H_OpMod;									
	HtgLmt					: FB_BA_HtgLmt;							
	TFlCtrl					: FB_BA_PID;
	GeneralSettings			: FB_BA_RawSubscriber;		
	stGeneralSettings		: ST_BA_GeneralSettings;	
END_VAR
VAR
	PlantLock				: FB_BA_PlantLock := (iParent := THIS^);
	
END_VAR
VAR // added by the converter: edge detectors and wires of the graphical bodies
    _w1 : ANY;
END_VAR

// note: 14 stored wires end on pins the file does not list and are not shown
SUPER^(); // FB_BA_View
GeneralSettings(xData := stGeneralSettings); // FB_BA_RawSubscriber
TFl(); // FB_BA_SensorAnalog_IO
TRt(); // FB_BA_SensorAnalog_IO
PlantLock(); // FB_BA_PlantLock
_w1 := PlantLock.bPrioHigh OR PlantLock.bPrioMedium;
HtgLmt(fIn := stGeneralSettings.fTWthDamped); // FB_BA_HtgLmt
OpMod(bDst := _w1, bHtgLmt := HtgLmt.bQ, bTWthLowLimit := stGeneralSettings.bTWthLowLimit); // FB_BA_H_OpMod
bRls := OpMod.bRls;
eOpMod := OpMod.eOpMod;
Sp(
    eOpMod := eOpMod,
    fSpFrstProtec := stGeneralSettings.fFrostProtectionSetpoint,
    fTWthDamp := stGeneralSettings.fTWthDamped); // FB_BA_H_HtgCir_Sp
fSp := Sp.fSpFlWT;
TFlCtrl(bEn := OpMod.bRls, fW := fSp, fX := TFl.fPresentValue); // FB_BA_PID
Pu(
    bEnSfty := PlantLock.bPrioHigh,
    bValSfty := FALSE,
    bEnCrit := PlantLock.bPrioMedium,
    bValCrit := FALSE,
    bEnPgm := OpMod.bRls,
    bValPgm := TRUE,
    bAblkLock := fVlv >= 10.0); // FB_BA_Pu1st
bPu := Pu.bCmd;
Vlv(
    bEnSfty := PlantLock.bPrioHigh,
    fValSfty := 0,
    bEnCrit := PlantLock.bPrioMedium,
    fValCrit := 0,
    bEnPgm := OpMod.bRls,
    fValPgm := TFlCtrl.fY,
    bAblkLock := Pu.bCmd); // FB_BA_Vlv
fVlv := Vlv.fPresentValue;

METHOD FB_init : BOOL
VAR_INPUT
	bInitRetains : BOOL; // if TRUE, the retain variables are initialized (warm start / cold start)
	bInCopyCode : BOOL;  // if TRUE, the instance afterwards gets moved into the copy code (online change)
END_VAR
TFl.iParent								:= THIS^;		
TFl.iLabel 								:= LblCmpHeating.H_HtgCir_TFl;	
TFl.sObjectName							:= '{Idx=01}';	
TFl.eDPADMode							:= E_BA_DPADMode.eInclude;																																	
TFl.MV.eUnit							:= E_BA_Unit.eTemperature_DegreesCelsius;
TFl.MV.fResolution 						:= 0.01;
TFl.MV.fScaleOffset 					:= 0; 
TFl.MV.bEventDetectionEnable			:= TRUE;
TFl.MV.eEnPlantLock						:= E_BA_LockPriority.eMedium;

TRt.iParent								:= THIS^;		
TRt.iLabel 								:= LblCmpHeating.H_HtgCir_TRt;	
TRt.sObjectName							:= '{Idx=01}';														
TRt.eDPADMode							:= E_BA_DPADMode.eInclude;																																	
TRt.MV.eUnit							:= E_BA_Unit.eTemperature_DegreesCelsius;
TRt.MV.fResolution 						:= 0.01;
TRt.MV.fScaleOffset 					:= 0;  
TRt.MV.bEventDetectionEnable			:= TRUE;
TRt.MV.eEnPlantLock						:= E_BA_LockPriority.eNoLock;
				
Vlv.iParent								:= THIS^;	
Vlv.iLabel								:= LblCmpHeating.H_HtgCir_Vlv;
Vlv.sObjectName							:= '{Idx=01}';										 
Vlv.eDPADMode							:= E_BA_DPADMode.eInclude;									
				
Pu.iParent								:= THIS^;
Pu.iLabel								:= LblCmpHeating.H_HtgCir_Pu;
Pu.sObjectName							:= '{Idx=01}';										 
Pu.eDPADMode							:= E_BA_DPADMode.eInclude;	
Pu.Dst.bEventDetectionEnable			:= TRUE;			
				
Sp.iParent								:= THIS^;	
Sp.iLabel								:= LblCmpHeating.H_HtgCir_Sp;
Sp.sObjectName							:= '{Idx=01}';										 
Sp.eDPADMode							:= E_BA_DPADMode.eInclude;												
				
OpMod.iParent							:= THIS^;	
OpMod.iLabel							:= LblCmpHeating.H_HtgCir_OpMod;
OpMod.sObjectName						:= '{Idx=01}';										 
OpMod.eDPADMode							:= E_BA_DPADMode.eInclude;									
				
HtgLmt.iParent							:= THIS^;	
HtgLmt.iLabel							:= LblCmpHeating.H_HtgCir_HtgLmt;
HtgLmt.sObjectName						:= '{Idx=01}';										 
HtgLmt.eDPADMode						:= E_BA_DPADMode.eInclude;

TFlCtrl.iParent							:= THIS^;
TFlCtrl.iLabel							:= LblCmpHeating.H_HtgCir_TFlCtrl;
TFlCtrl.sObjectName						:= '{Idx=01}';
TFlCtrl.eDPADMode						:= E_BA_DPADMode.eInclude;																																	
TFlCtrl.Ctrl.eOutputUnit				:= E_BA_Unit.eOther_Percent;
TFlCtrl.Ctrl.eActionRm					:= E_BA_Action.eReverse;
TFlCtrl.Ctrl.fMinOutputRm				:= 0;
TFlCtrl.Ctrl.fMaxOutputRm				:= 100;
TFlCtrl.Ctrl.fProportionalConstant		:= 3;
TFlCtrl.Ctrl.fIntegralConstant			:= 180;

GeneralSettings.Subject					:= Site.GeneralSettings_Subject;
GeneralSettings.sTarget					:= Site.GeneralSettings_NetId;
END_METHOD

END_FUNCTION_BLOCK

// ---- Templates/POUs/Universal/Sensor/FB_BA_SensorAnalog_IO.TcPOU
{region '#Template'}
	{attribute 'Version' := '1.0.0.0'}
	{attribute 'Tags' := '"LCID": "1031", "Text": "Universal, Sensor, AI"'}
	{attribute 'Tags' := '"LCID": "1033", "Text": "Universal, Sensor, AI"'}
	{attribute 'Description' := '"LCID": "1031", "Text": "AI mit IO"'}
	{attribute 'Description' := '"LCID": "1033", "Text": "AI with IO"'}
{endregion}	 
FUNCTION_BLOCK FB_BA_SensorAnalog_IO EXTENDS FB_BA_View
VAR_INPUT
END_VAR
VAR_INPUT CONSTANT
	MV					: FB_BA_AI_IO;		
END_VAR
VAR_OUTPUT
	fPresentValue		: REAL;
	bEvent				: BOOL;
	eEventState			: E_BA_EventState;	
END_VAR
VAR
END_VAR

SUPER^(); // FB_BA_View
MV(); // FB_BA_AI_IO
bEvent := MV.bEvent;
eEventState := MV.eEventState;
fPresentValue := MV.fPresentValue;

METHOD FB_init : BOOL
VAR_INPUT
	bInitRetains : BOOL; // if TRUE, the retain variables are initialized (warm start / cold start)
	bInCopyCode : BOOL;  // if TRUE, the instance afterwards gets moved into the copy code (online change)
END_VAR
MV.iParent						:= THIS^;		
MV.iLabel 						:= LblUniFieldDevice.SensorAnalog_MV;
MV.sObjectName					:= '{Idx=01}';
MV.sDeviceType					:= '';
MV.bEnOutOfService				:= FALSE;
MV.eUnit						:= E_BA_Unit.eTemperature_DegreesCelsius;
MV.fResolution 					:= 0.01;
MV.fScaleOffset 				:= 0; 	
MV.fCOVIncrement				:= BA2_Param.fDefCOVIncrement;
MV.nEventClassID				:= EventClasses.AlarmTechnicalExtended;
MV.stTimeDelay.nToNormal		:= BA2_Param.nDefTimeDelay_ToNormal;
MV.stTimeDelay.nToAbnormal		:= BA2_Param.nDefTimeDelay_ToAbnormal;
MV.stHighLimit.bEnable			:= FALSE;
MV.stHighLimit.fValue			:= 0.0;		
MV.stLowLimit.bEnable			:= FALSE;
MV.stLowLimit.fValue			:= 0.0;
MV.fLimitDeadband 				:= BA2_Param.fDefLimitDeadband;
MV.bAcknowledgeRm				:= FALSE;	
MV.aEventTransitionText[1]		:= txtEvent_Exceeded;
MV.aEventTransitionText[2]		:= txtEvent_Disturb;
MV.aEventTransitionText[3]		:= txtEvent_Normal;
MV.bEventDetectionEnable		:= TRUE;
MV.eEnPlantLock					:= E_BA_LockPriority.eNoLock;
END_METHOD

END_FUNCTION_BLOCK

// ---- Templates/POUs/Universal/Valve/FB_BA_Vlv.TcPOU
{region '#Template'}
	{attribute 'Version' := '1.0.0.0'}
	{attribute 'Tags' := '"LCID": "1031", "Text": "Universal, Valve"'}
	{attribute 'Tags' := '"LCID": "1033", "Text": "Universal, Valve"'}
	{attribute 'Description' := '"LCID": "1031", "Text": "Ventil analog"'}
	{attribute 'Description' := '"LCID": "1033", "Text": "Valve analog"'}
{endregion}		 
FUNCTION_BLOCK FB_BA_Vlv EXTENDS FB_BA_ActuatorAnalog
VAR_INPUT
	bAblkLock				: BOOL;
END_VAR
VAR_OUTPUT
END_VAR
VAR_INPUT CONSTANT
	Ablk					: FB_BA_AntiBlocking;	
	Fdb						: FB_BA_AI_IO;		 
END_VAR

Ablk(bFdb := fPresentValue >= 30.0, bLock := bAblkLock); // FB_BA_AntiBlocking
SUPER^(bEnPgm := Ablk.bQ OR bEnPgm, fValPgm := SEL(Ablk.bQ, fValPgm, 100)); // FB_BA_ActuatorAnalog
Fdb(); // FB_BA_AI_IO

METHOD FB_init : BOOL
VAR_INPUT
	bInitRetains : BOOL; // if TRUE, the retain variables are initialized (warm start / cold start)
	bInCopyCode : BOOL;  // if TRUE, the instance afterwards gets moved into the copy code (online change)
END_VAR
Ablk.iParent					:= THIS^;	
Ablk.iLabel						:= LblUniFieldDevice.Valve_Ablk;
Ablk.sObjectName				:= '{Idx=01}';																	
Ablk.eDPADMode					:= E_BA_DPADMode.eIncludeDescription;	

Fdb.iParent						:= THIS^;		
Fdb.iLabel 						:= LblUniFieldDevice.Valve_Fdb;
Fdb.sObjectName					:= '{Idx=01}';
Fdb.sDeviceType					:= '';
Fdb.bEnOutOfService				:= FALSE;
Fdb.eUnit						:= E_BA_Unit.eOther_Percent;
Fdb.fResolution 				:= 0.03051851;
Fdb.fScaleOffset 				:= 0; 	
Fdb.fCOVIncrement				:= BA2_Param.fDefCOVIncrement;
Fdb.nEventClassID				:= EventClasses.OtherSimple;
Fdb.stTimeDelay.nToNormal		:= BA2_Param.nDefTimeDelay_ToNormal;
Fdb.stTimeDelay.nToAbnormal		:= BA2_Param.nDefTimeDelay_ToAbnormal;
Fdb.stHighLimit.bEnable			:= FALSE;
Fdb.stHighLimit.fValue			:= 0.0;		
Fdb.stLowLimit.bEnable			:= FALSE;
Fdb.stLowLimit.fValue			:= 0.0;
Fdb.fLimitDeadband 				:= BA2_Param.fDefLimitDeadband;
Fdb.bAcknowledgeRm				:= FALSE;	
Fdb.aEventTransitionText[1]		:= txtEvent_Exceeded;
Fdb.aEventTransitionText[2]		:= txtEvent_Disturb;
Fdb.aEventTransitionText[3]		:= txtEvent_Normal;
Fdb.bEventDetectionEnable		:= FALSE;
Fdb.eEnPlantLock				:= E_BA_LockPriority.eNoLock;
END_METHOD

END_FUNCTION_BLOCK

// ---- Templates/POUs/Universal/Aggregat/Analog/FB_BA_ActuatorAnalog.TcPOU
{region '#Template'}
	{attribute 'Version' := '1.0.0.0'}
	{attribute 'Tags' := '"LCID": "1031", "Text": "Universal, Analog, Aggregate"'}
	{attribute 'Tags' := '"LCID": "1033", "Text": "Universal, Analog, Aggregate"'}
	{attribute 'Description' := '"LCID": "1031", "Text": "Aktor analog"'}
	{attribute 'Description' := '"LCID": "1033", "Text": "Actuator analog"'}
{endregion}
FUNCTION_BLOCK FB_BA_ActuatorAnalog EXTENDS FB_BA_AggregateA
VAR_OUTPUT
	fPresentValue			: REAL;
END_VAR
VAR_INPUT CONSTANT
	Mdlt					: FB_BA_AO_IO;
END_VAR
VAR
END_VAR

SUPER^(); // FB_BA_AggregateA
Mdlt(
    bEnSfty := bEnSfty,
    fValSfty := SUPER^.fActiveVal,
    bEnCrit := bEnCrit,
    fValCrit := SUPER^.fActiveVal,
    bEnPgm := bEnPgm,
    fValPgm := SUPER^.fActiveVal); // FB_BA_AO_IO
fPresentValue := Mdlt.fPresentValue;

METHOD FB_init : BOOL
VAR_INPUT
	bInitRetains : BOOL; // if TRUE, the retain variables are initialized (warm start / cold start)
	bInCopyCode : BOOL;  // if TRUE, the instance afterwards gets moved into the copy code (online change)
END_VAR
Mdlt.iParent					:= THIS^;
Mdlt.iLabel						:= LblUniFieldDevice.Aggregat_Mdlt;	
Mdlt.sObjectName				:= '{Idx=01}';
Mdlt.sDeviceType				:= '';
Mdlt.bEnOutOfService			:= FALSE;
Mdlt.eOverriddenPolarity		:= E_BA_Polarity.eNormal;
Mdlt.eUnit						:= E_BA_Unit.eOther_Percent;
Mdlt.fResolution 				:= 0.003051851;
Mdlt.fScaleOffset 				:= 0;
Mdlt.fCOVIncrement				:= BA2_Param.fDefCOVIncrement;
Mdlt.bEnManualRm				:= FALSE;	//	Priority  8	
Mdlt.fValManualRm				:= 0.0;		//	Priority  8
Mdlt.fDefaultValue				:= 0.0;	
Mdlt.nEventClassID				:= EventClasses.NotificationSimple;
Mdlt.stTimeDelay.nToNormal		:= BA2_Param.nDefTimeDelay_ToNormal;
Mdlt.stTimeDelay.nToAbnormal	:= BA2_Param.nDefTimeDelay_ToAbnormal;
Mdlt.stHighLimit.bEnable		:= FALSE;
Mdlt.stHighLimit.fValue			:= 0.0;		
Mdlt.stLowLimit.bEnable			:= FALSE;
Mdlt.stLowLimit.fValue			:= 0.0;
Mdlt.fLimitDeadband 			:= BA2_Param.fDefLimitDeadband;
Mdlt.bAcknowledgeRm				:= FALSE;	
Mdlt.aEventTransitionText[1]	:= txtEvent_Disturb;
Mdlt.aEventTransitionText[2]	:= txtEvent_None;
Mdlt.aEventTransitionText[3]	:= txtEvent_Normal;
Mdlt.bEventDetectionEnable		:= FALSE;
Mdlt.eEnPlantLock				:= E_BA_LockPriority.eNoLock;
END_METHOD

END_FUNCTION_BLOCK

// ---- Templates/POUs/Universal/Control/AntiBlocking/FB_BA_AntiBlocking.TcPOU
{region '#Template'}
	{attribute 'Version' := '1.0.0.0'}
	{attribute 'Tags' := '"LCID": "1031", "Text": "Universal, Control, Antiblockierschutz"'}
	{attribute 'Tags' := '"LCID": "1033", "Text": "Universal, Control, Anti-blocking protection"'}
	{attribute 'Description' := '"LCID": "1031", "Text": "Antiblockierschutz"'}
	{attribute 'Description' := '"LCID": "1033", "Text": "Anti-blocking protection"'}
{endregion}
FUNCTION_BLOCK FB_BA_AntiBlocking EXTENDS FB_BA_View
VAR_INPUT
	bFdb					: BOOL;	
	bExtReq					: BOOL;
	bLock					: BOOL;
END_VAR
VAR_OUTPUT
	bQ						: BOOL;
END_VAR
VAR_INPUT CONSTANT PERSISTENT
	{attribute 'parameterCategory' := 'Operation'}
	bEn : BOOL := TRUE;
END_VAR
VAR_INPUT CONSTANT
	IdlePrd					: FB_BA_AV_Op;									 
	ImpulseLength			: FB_BA_AV_Op;
END_VAR	
VAR		
	AblkFnct				: FB_BA_AntBlkg;
	tonEn					: TON;
END_VAR

SUPER^(); // FB_BA_View
IdlePrd(); // FB_BA_AV_Op
AblkFnct.nOffMin := MAX(TO_UDINT(IdlePrd.fPresentValue) * 3600, 60);
ImpulseLength(); // FB_BA_AV_Op
AblkFnct.nImplLngt := MAX(TO_UDINT(ImpulseLength.fPresentValue), 10);
tonEn(IN := bEn, PT := T#2s); // TON
AblkFnct(bEn := tonEn.Q, bFdb := bFdb, bExtReq := bExtReq, bLock := bLock); // FB_BA_AntBlkg
bQ := AblkFnct.bQ;

METHOD FB_init : BOOL
VAR_INPUT
	bInitRetains : BOOL; // if TRUE, the retain variables are initialized (warm start / cold start)
	bInCopyCode : BOOL;  // if TRUE, the instance afterwards gets moved into the copy code (online change)
END_VAR
IdlePrd.iParent					:= THIS^;
IdlePrd.iLabel					:= LblUniControl.AntiBlocking_IdlePeriod;	
IdlePrd.sObjectName				:= '{Idx=01}';								 	 
IdlePrd.eUnit 					:= E_BA_Unit.eTime_Hours;								 
IdlePrd.fValueRm				:= 168;
IdlePrd.fCOVIncrement			:= BA2_Param.fDefCOVIncrement;
														 
ImpulseLength.iParent			:= THIS^;
ImpulseLength.iLabel			:= LblUniControl.AntiBlocking_ImpulsLength;	
ImpulseLength.sObjectName		:= '{Idx=01}';								 	 
ImpulseLength.eUnit 			:= E_BA_Unit.eTime_Seconds;								 
ImpulseLength.fValueRm			:= 240;					
ImpulseLength.fCOVIncrement		:= BA2_Param.fDefCOVIncrement;
END_METHOD

END_FUNCTION_BLOCK

// ---- Templates/POUs/Universal/Pump/1st/FB_BA_Pu1st.TcPOU
{region '#Template'}
	{attribute 'Version' := '1.0.0.0'}
	{attribute 'Tags' := '"LCID": "1031", "Text": "Universal, Pump"'}
	{attribute 'Tags' := '"LCID": "1033", "Text": "Universal, Pump"'}
	{attribute 'Description' := '"LCID": "1031", "Text": "Pumpe 1 stufig"'}
	{attribute 'Description' := '"LCID": "1033", "Text": "Pump 1 stage"'}
{endregion}	 
FUNCTION_BLOCK FB_BA_Pu1st EXTENDS FB_BA_Mot1st
VAR_INPUT
	bAblkLock				: BOOL;	
END_VAR
VAR_INPUT CONSTANT
	DlyOff					: FB_BA_DlyOff;								
	Ablk					: FB_BA_AntiBlocking;							
END_VAR
VAR
	PrioSwiPgm				: FB_BA_PrioSwi_B04;
END_VAR

DlyOff(bVal := bEnPgm AND bValPgm); // FB_BA_DlyOff
// parameter Ablk.sObjectName := '[Idx=01]'
Ablk(bFdb := bCmd, bLock := bAblkLock); // FB_BA_AntiBlocking
PrioSwiPgm(bEn03 := DlyOff.bQ, bVal03 := TRUE, bEn04 := Ablk.bQ, bVal04 := TRUE); // FB_BA_PrioSwi_B04
SUPER^(bEnPgm := PrioSwiPgm.bQ, bValPgm := PrioSwiPgm.bVal); // FB_BA_Mot1st

METHOD FB_init : BOOL
VAR_INPUT
	bInitRetains : BOOL; // if TRUE, the retain variables are initialized (warm start / cold start)
	bInCopyCode : BOOL;  // if TRUE, the instance afterwards gets moved into the copy code (online change)
END_VAR
DlyOff.iParent			:= THIS^;	
DlyOff.iLabel			:= LblUniFieldDevice.Pump_DlyOff;
DlyOff.sObjectName		:= '{Idx=01}';									
DlyOff.eDPADMode		:= E_BA_DPADMode.eIncludeDescription;

Ablk.iParent			:= THIS^;	
Ablk.iLabel				:= LblUniFieldDevice.Pump_Ablk;
Ablk.sObjectName		:= '{Idx=01}';																	
Ablk.eDPADMode			:= E_BA_DPADMode.eIncludeDescription;
END_METHOD

END_FUNCTION_BLOCK

// ---- Templates/POUs/Universal/Motor/1st/FB_BA_Mot1st.TcPOU
{region '#Template'}
	{attribute 'Version' := '1.0.0.0'}
	{attribute 'Tags' := '"LCID": "1031", "Text": "Universal, Motor, Aggregate"'}
	{attribute 'Tags' := '"LCID": "1033", "Text": "Universal, Motor, Aggregate"'}
	{attribute 'Description' := '"LCID": "1031", "Text": "Motor 1 stufig"'}
	{attribute 'Description' := '"LCID": "1033", "Text": "Motor 1 stage"'}
{endregion}	 
FUNCTION_BLOCK FB_BA_Mot1st EXTENDS FB_BA_AggregateB
VAR_OUTPUT
	bCmd		: BOOL;
END_VAR
VAR_INPUT CONSTANT
	Dst			: FB_BA_BI_IO;
	
	Cmd			: FB_BA_BO_IO;							
END_VAR

Dst(); // FB_BA_BI_IO
SUPER^(); // FB_BA_AggregateB
Cmd(
    bEnSfty := bEnSfty,
    bValSfty := SUPER^.bActiveVal,
    bEnCrit := bEnCrit,
    bValCrit := SUPER^.bActiveVal,
    bEnPgm := bEnPgm,
    bValPgm := SUPER^.bActiveVal); // FB_BA_BO_IO
bCmd := Cmd.bPresentValue;

METHOD FB_init : BOOL
VAR_INPUT
	bInitRetains : BOOL; // if TRUE, the retain variables are initialized (warm start / cold start)
	bInCopyCode : BOOL;  // if TRUE, the instance afterwards gets moved into the copy code (online change)
END_VAR
Dst.iParent							:= THIS^;
Dst.iLabel							:= LblUniFieldDevice.Motor_Dst;	
Dst.sObjectName						:= '{Idx=01}';	
Dst.sDeviceType						:= '';
Dst.bEnOutOfService					:= FALSE;
Dst.ePolarity						:= E_BA_Polarity.eReverse;
Dst.sActiveText 					:= txtEvent_Triggered;
Dst.sInactiveText 					:= txtEvent_Normal;
Dst.nStateChangeCount				:= 0;
Dst.nActiveTimeElapsed				:= 0;
Dst.nEventClassID					:= EventClasses.AlarmTechnicalExtended;
Dst.stTimeDelay.nToNormal			:= BA2_Param.nDefTimeDelay_ToNormal;
Dst.stTimeDelay.nToAbnormal			:= BA2_Param.nDefTimeDelay_ToAbnormal;
Dst.bAlarmValue						:= TRUE;
Dst.bAcknowledgeRm					:= FALSE;	
Dst.aEventTransitionText[1]			:= txtEvent_Triggered;
Dst.aEventTransitionText[2]			:= txtEvent_Error;
Dst.aEventTransitionText[3]			:= txtEvent_Normal;
Dst.bEventDetectionEnable			:= TRUE;
Dst.eEnPlantLock					:= E_BA_LockPriority.eLocalMedium;

Cmd.iParent							:= THIS^;
Cmd.iLabel							:= LblUniFieldDevice.Motor_Cmd;			
Cmd.sObjectName						:= '{Idx=01}';
Cmd.sDeviceType						:= '';	
Cmd.ePolarity						:= E_BA_Polarity.eNormal;
Cmd.eFeedbackPolarity				:= E_BA_Polarity.eNormal;
Cmd.eOverriddenPolarity				:= E_BA_Polarity.eReverse;
Cmd.sActiveText 					:= txtEvent_On;
Cmd.sInactiveText 					:= txtEvent_Off;
Cmd.nStateChangeCount				:= 0;
Cmd.nActiveTimeElapsed				:= 0;
Cmd.nMinimumOnTime					:= 0;
Cmd.nMinimumOffTime					:= 0;
Cmd.bEnManualRm						:= FALSE;	//	Priority  8	
Cmd.bValManualRm					:= FALSE;	//	Priority  8
Cmd.bDefaultValue					:= FALSE;
Cmd.nEventClassID					:= EventClasses.DisturbanceExtended;
Cmd.stTimeDelay.nToNormal			:= BA2_Param.nDefTimeDelay_ToNormal;
Cmd.stTimeDelay.nToAbnormal			:= BA2_Param.nDefTimeDelay_ToAbnormal;
Cmd.bAcknowledgeRm					:= FALSE;		
Cmd.aEventTransitionText[1]			:= txtEvent_Disturb;
Cmd.aEventTransitionText[2]			:= txtEvent_None;
Cmd.aEventTransitionText[3]			:= txtEvent_Normal;
Cmd.bEventDetectionEnable			:= FALSE;
Cmd.eEnPlantLock					:= E_BA_LockPriority.eNoLock;
END_METHOD

END_FUNCTION_BLOCK

// ---- Templates/POUs/Universal/Control/TimeDelay/FB_BA_DlyOff.TcPOU
{region '#Template'}
	{attribute 'Version' := '1.0.0.0'}
	{attribute 'Tags' := '"LCID": "1031", "Text": "Universal, Control, Timer"'}
	{attribute 'Tags' := '"LCID": "1033", "Text": "Universal, Control, Timer"'}
	{attribute 'Description' := '"LCID": "1031", "Text": "Zeitglied Ausschaltverzögert"'}
	{attribute 'Description' := '"LCID": "1033", "Text": "Timer switch-off delayed"'}
{endregion}
FUNCTION_BLOCK FB_BA_DlyOff EXTENDS FB_BA_View
VAR_INPUT
	bVal					: BOOL;	
END_VAR
VAR_OUTPUT
	bQ						: BOOL;	
	nRT						: UDINT;// Restzeit [s] // remaining time [s]
END_VAR
VAR_INPUT CONSTANT
	TiDly					: FB_BA_AV_Op;			
END_VAR	
VAR	
	tofDlyOff				: TOF;
END_VAR
VAR // added by the converter: edge detectors and wires of the graphical bodies
    _w1, _w2 : ANY;
END_VAR

SUPER^(); // FB_BA_View
TiDly(); // FB_BA_AV_Op
_w1 := F_BA_RealToTiSec(fSec := TiDly.fPresentValue);
tofDlyOff(IN := bVal, PT := _w1); // TOF
bQ := tofDlyOff.Q;
_w2 := F_BA_RemSecsTof(tofTimer := tofDlyOff);
nRT := _w2;

METHOD FB_init : BOOL
VAR_INPUT
	bInitRetains : BOOL; // if TRUE, the retain variables are initialized (warm start / cold start)
	bInCopyCode : BOOL;  // if TRUE, the instance afterwards gets moved into the copy code (online change)
END_VAR
TiDly.iParent			:= THIS^;
TiDly.iLabel			:= LblUniControl.DelayOff_TiDly;		 
TiDly.sObjectName		:= '{Idx=01}';								 	 
TiDly.eUnit 			:= E_BA_Unit.eTime_Seconds;								 
TiDly.fValueRm			:= 0;															 
TiDly.fCOVIncrement		:= BA2_Param.fDefCOVIncrement;
END_METHOD

END_FUNCTION_BLOCK

// ---- Templates/POUs/Trade/HeatingSystem/Setpoint/FB_BA_H_HtgCir_Sp.TcPOU
{region '#Template'}
	{attribute 'Version' := '1.0.0.0'}
	{attribute 'Tags' := '"LCID": "1031", "Text": "H, Heating circuit, HtgCir, Setpoint"'}
	{attribute 'Tags' := '"LCID": "1033", "Text": "H, Heating circuit, HtgCir, Setpoint"'}
	{attribute 'Description' := '"LCID": "1031", "Text": "Sollwert Heizkreis"'}
	{attribute 'Description' := '"LCID": "1033", "Text": "Setpoint heating circuit"'}
{endregion}
FUNCTION_BLOCK FB_BA_H_HtgCir_Sp EXTENDS FB_BA_View
VAR_INPUT
	eOpMod					: E_BA_EnergyLvl;
	fSpFrstProtec			: REAL;
	fTWthDamp				: REAL;
END_VAR
VAR_OUTPUT
	fSpFlWT							: REAL;
END_VAR
VAR_INPUT CONSTANT
	NgtOffs					: FB_BA_AV_Op;	
	SpFlWT					: FB_BA_AV_Op;		
	HtgCrv					: FB_BA_Scale_04; 
END_VAR
VAR
	PrioSwi					: FB_BA_MMUX_R04;
END_VAR

// note: 1 stored wires end on pins the file does not list and are not shown
SUPER^(); // FB_BA_View
NgtOffs(); // FB_BA_AV_Op
HtgCrv(fX := fTWthDamp); // FB_BA_Scale_04
PrioSwi(
    bEn := TRUE,
    nSel := eOpMod,
    nEn01 := E_BA_EnergyLvl.eComfort,
    fVal01 := HtgCrv.fY,
    nEn02 := E_BA_EnergyLvl.eEconomy,
    fVal02 := HtgCrv.fY - ABS(NgtOffs.fPresentValue),
    nEn03 := E_BA_EnergyLvl.eProtection,
    fVal03 := fSpFrstProtec); // FB_BA_MMUX_R04
SpFlWT(fValuePgm := PrioSwi.fVal); // FB_BA_AV_Op
fSpFlWT := SpFlWT.fPresentValue;

METHOD FB_init : BOOL
VAR_INPUT
	bInitRetains : BOOL; // if TRUE, the retain variables are initialized (warm start / cold start)
	bInCopyCode : BOOL;  // if TRUE, the instance afterwards gets moved into the copy code (online change)
END_VAR
NgtOffs.iParent				:= THIS^;
NgtOffs.iLabel				:= LblCmpHeating.H_HtgCir_Sp_NgtOffs;		 
NgtOffs.sObjectName			:= '{Idx=01}';
NgtOffs.eUnit				:= E_BA_Unit.eTemperature_DegreesCelsius;  
NgtOffs.fValueRm			:= 8.0;
NgtOffs.fCOVIncrement	:= BA2_Param.fDefCOVIncrement;							

SpFlWT.iParent				:= THIS^;
SpFlWT.iLabel				:= LblCmpHeating.H_HtgCir_Sp_SpFlWT;		 
SpFlWT.sObjectName			:= '{Idx=01}';
SpFlWT.eUnit				:= E_BA_Unit.eTemperature_DegreesCelsius;  
SpFlWT.fCOVIncrement		:= BA2_Param.fDefCOVIncrement;							

HtgCrv.iParent				:= THIS^;										
HtgCrv.iLabel				:= LblCmpHeating.H_HtgCir_Sp_HtgCrv;
HtgCrv.sObjectName			:= '{Idx=01}';										 
HtgCrv.eDPADMode			:= E_BA_DPADMode.eIncludeDescription; 
HtgCrv.X1.fValueRm			:= 15.0;
HtgCrv.X2.fValueRm			:= 0.0;
HtgCrv.X3.fValueRm			:= -10.0;
HtgCrv.X4.fValueRm			:= -20.0;
HtgCrv.Y1.fValueRm			:= 25.0;
HtgCrv.Y2.fValueRm			:= 40.0;
HtgCrv.Y3.fValueRm			:= 55.0;
HtgCrv.Y4.fValueRm			:= 65.0;
HtgCrv.YMin.fValueRm		:= 5.0;
HtgCrv.YMax.fValueRm		:= 80.0;
END_METHOD

END_FUNCTION_BLOCK

// ---- Templates/POUs/Universal/Control/Scale/FB_BA_Scale_04.TcPOU
{region '#Template'}
	{attribute 'Version' := '1.0.0.0'}
	{attribute 'Tags' := '"LCID": "1031", "Text": "Universal, Control, Scaling"'}
	{attribute 'Tags' := '"LCID": "1033", "Text": "Universal, Control, Scaling"'}
	{attribute 'Description' := '"LCID": "1031", "Text": "Skalierung"'}
	{attribute 'Description' := '"LCID": "1033", "Text": "Scaling"'}
{endregion}
FUNCTION_BLOCK FB_BA_Scale_04 EXTENDS FB_BA_View
VAR_INPUT
	fX			: REAL;
END_VAR
VAR_OUTPUT
	fY			: REAL;
END_VAR
VAR_INPUT CONSTANT
	X1			: FB_BA_AV_Op;	
	X2			: FB_BA_AV_Op;	
	X3			: FB_BA_AV_Op;	
	X4			: FB_BA_AV_Op;	
	Y1			: FB_BA_AV_Op;	
	Y2			: FB_BA_AV_Op;
	Y3			: FB_BA_AV_Op;
	Y4			: FB_BA_AV_Op;
	YMin		: FB_BA_AV_Op;			
	YMax		: FB_BA_AV_Op;			
	Y			: FB_BA_AV_Op;		
END_VAR
VAR		
	Scale		: FB_BA_Chrct04;
END_VAR

SUPER^(); // FB_BA_View
X1(); // FB_BA_AV_Op
X2(); // FB_BA_AV_Op
X3(); // FB_BA_AV_Op
X4(); // FB_BA_AV_Op
Y1(); // FB_BA_AV_Op
Y2(); // FB_BA_AV_Op
Y3(); // FB_BA_AV_Op
Y4(); // FB_BA_AV_Op
Ymin(); // FB_BA_AV_Op
YMax(); // FB_BA_AV_Op
Scale(
    fX := fX,
    fX01 := X1.fPresentValue,
    fX02 := X2.fPresentValue,
    fX03 := X3.fPresentValue,
    fX04 := X4.fPresentValue,
    fY01 := Y1.fPresentValue,
    fY02 := Y2.fPresentValue,
    fY03 := Y3.fPresentValue,
    fY04 := Y4.fPresentValue,
    fYMin := Ymin.fPresentValue,
    fYMax := YMax.fPresentValue); // FB_BA_Chrct04
Y(fValuePgm := Scale.fCalcVal); // FB_BA_AV_Op
fY := Y.fPresentValue;

METHOD FB_init : BOOL
VAR_INPUT
	bInitRetains : BOOL; // if TRUE, the retain variables are initialized (warm start / cold start)
	bInCopyCode : BOOL;  // if TRUE, the instance afterwards gets moved into the copy code (online change)
END_VAR
X1.iParent			:= THIS^;
X1.iLabel			:= LblUniControl.Scale_X01;	
X1.sObjectName		:= '{Idx=01}';								 	 
X1.eUnit			:= E_BA_Unit.eTemperature_DegreesCelsius;						 	 
X1.fValueRm			:= 15.0;
X1.fCOVIncrement	:= BA2_Param.fDefCOVIncrement;		

X2.iParent			:= THIS^;
X2.iLabel			:= LblUniControl.Scale_X02;							
X2.sObjectName		:= '{Idx=02}';								 	 
X2.eUnit			:= E_BA_Unit.eTemperature_DegreesCelsius;						 	 
X2.fValueRm			:= 0.0;
X2.fCOVIncrement	:= BA2_Param.fDefCOVIncrement;		

X3.iParent			:= THIS^;
X3.iLabel			:= LblUniControl.Scale_X03;	 						
X3.sObjectName		:= '{Idx=03}';								 	 
X3.eUnit			:= E_BA_Unit.eTemperature_DegreesCelsius;						 	 
X3.fValueRm			:= -10.0;
X3.fCOVIncrement	:= BA2_Param.fDefCOVIncrement;		

X4.iParent			:= THIS^;
X4.iLabel			:= LblUniControl.Scale_X04;						
X4.sObjectName		:= '{Idx=04}';								 	 
X4.eUnit			:= E_BA_Unit.eTemperature_DegreesCelsius;						 	 
X4.fValueRm			:= -20.0;
X4.fCOVIncrement	:= BA2_Param.fDefCOVIncrement;		

Y1.iParent			:= THIS^;
Y1.iLabel			:= LblUniControl.Scale_Y01;							
Y1.sObjectName		:= '{Idx=01}';								 	 
Y1.eUnit			:= E_BA_Unit.eTemperature_DegreesCelsius;						 	 
Y1.fValueRm			:= 25.0;
Y1.fCOVIncrement	:= BA2_Param.fDefCOVIncrement;		

Y2.iParent			:= THIS^;
Y2.iLabel			:= LblUniControl.Scale_Y02;				
Y2.sObjectName		:= '{Idx=02}';								 	 
Y2.eUnit			:= E_BA_Unit.eTemperature_DegreesCelsius;						 	 
Y2.fValueRm			:= 40.0;
Y2.fCOVIncrement	:= BA2_Param.fDefCOVIncrement;		

Y3.iParent			:= THIS^;
Y3.iLabel			:= LblUniControl.Scale_Y03;				
Y3.sObjectName		:= '{Idx=03}';								 	 
Y3.eUnit			:= E_BA_Unit.eTemperature_DegreesCelsius;						 	 
Y3.fValueRm			:= 55.0;
Y3.fCOVIncrement	:= BA2_Param.fDefCOVIncrement;		

Y4.iParent			:= THIS^;
Y4.iLabel			:= LblUniControl.Scale_Y04;				
Y4.sObjectName		:= '{Idx=04}';								 	 
Y4.eUnit			:= E_BA_Unit.eTemperature_DegreesCelsius;						 	 
Y4.fValueRm			:= 65.0;
Y4.fCOVIncrement	:= BA2_Param.fDefCOVIncrement;		

YMin.iParent		:= THIS^;
YMin.iLabel			:= LblUniControl.Scale_Ymin;		
YMin.sObjectName	:= '{Idx=01}';								 	 
YMin.eUnit			:= E_BA_Unit.eTemperature_DegreesCelsius;						 	 
YMin.fValueRm		:= 5.0;
YMin.fCOVIncrement	:= BA2_Param.fDefCOVIncrement;		

YMax.iParent		:= THIS^;
YMax.iLabel			:= LblUniControl.Scale_Ymax;			
YMax.sObjectName	:= '{Idx=01}';								 	 
YMax.eUnit			:= E_BA_Unit.eTemperature_DegreesCelsius;						 	 
YMax.fValueRm		:= 80.0;
YMax.fCOVIncrement	:= BA2_Param.fDefCOVIncrement;		

Y.iParent			:= THIS^;
Y.iLabel			:= LblUniControl.Scale_Y;				
Y.sObjectName		:= '{Idx=01}';								 	 
Y.eUnit				:= E_BA_Unit.eTemperature_DegreesCelsius;	
Y.fCOVIncrement		:= BA2_Param.fDefCOVIncrement;
END_METHOD

METHOD GetPoint : BOOL
VAR_INPUT
	nIndex		: INT;
END_VAR
VAR_OUTPUT
	fbObjectX	: I_BA_AnalogOpObject;
	fbObjectY	: I_BA_AnalogOpObject;
END_VAR
CASE (nIndex) OF
	1:
		fbObjectX := X1;
		fbObjectY := Y1;
	2:
		fbObjectX := X2;
		fbObjectY := Y2;
	3:
		fbObjectX := X3;
		fbObjectY := Y3;
	4:
		fbObjectX := X4;
		fbObjectY := Y4;
ELSE
	RETURN;
END_CASE

GetPoint := TRUE;
END_METHOD

END_FUNCTION_BLOCK

// ---- Templates/POUs/Trade/HeatingSystem/General/FB_BA_H_OpMod.TcPOU
{region '#Template'}
	{attribute 'Version' := '1.0.0.0'}
	{attribute 'Tags' := '"LCID": "1031", "Text": "H, General, HtgCir, Operating mode"'}
	{attribute 'Tags' := '"LCID": "1033", "Text": "H, General, HtgCir, Operating mode"'}
	{attribute 'Description' := '"LCID": "1031", "Text": "Betriebsart"'}
	{attribute 'Description' := '"LCID": "1033", "Text": "Operating mode"'}
{endregion}
FUNCTION_BLOCK FB_BA_H_OpMod EXTENDS FB_BA_View
VAR_INPUT
	bDst					: BOOL;
	bHtgLmt					: BOOL;
	bTWthLowLimit			: BOOL;
END_VAR
VAR_OUTPUT
	eOpMod					: E_BA_EnergyLvl;
	bRls					: BOOL;
END_VAR
VAR_INPUT CONSTANT
	OpModMan				: FB_BA_MV_Op;
	Sched					: FB_BA_SchedM;
	OpModPr					: FB_BA_MV_Op;								 
	Rls						: FB_BA_BV_Op;
END_VAR
VAR
	OpModSwi				: FB_BA_PrioSwi_UDI08;
	RlsMMux					: FB_BA_MMUX_B04;
END_VAR

SUPER^(); // FB_BA_View
OpModMan(); // FB_BA_MV_Op
Sched(); // FB_BA_SchedM
OpModSwi(
    bEn01 := bDst,
    nVal01 := E_BA_EnergyLvl.eProtection,
    bEn02 := OpModMan.nPresentValue = E_BA_EnergyLvlA.eProtection,
    nVal02 := E_BA_EnergyLvl.eProtection,
    bEn03 := OpModMan.nPresentValue = E_BA_EnergyLvlA.eEconomy,
    nVal03 := E_BA_EnergyLvl.eEconomy,
    bEn04 := OpModMan.nPresentValue = E_BA_EnergyLvlA.eComfort,
    nVal04 := E_BA_EnergyLvl.eComfort,
    bEn05 := NOT bHtgLmt,
    nVal05 := E_BA_EnergyLvl.eProtection,
    bEn06 := Sched.nPresentValue = E_BA_EnergyLvl.eProtection,
    nVal06 := E_BA_EnergyLvl.eProtection,
    bEn07 := Sched.nPresentValue = E_BA_EnergyLvl.eEconomy,
    nVal07 := E_BA_EnergyLvl.eEconomy,
    bEn08 := Sched.nPresentValue = E_BA_EnergyLvl.eComfort,
    nVal08 := E_BA_EnergyLvl.eComfort); // FB_BA_PrioSwi_UDI08
OpModPr(nValuePgm := OpModSwi.nVal); // FB_BA_MV_Op
eOpMod := OpModPr.nPresentValue;
RlsMMux(
    bEn := TRUE,
    nSel := eOpMod,
    nEn01 := E_BA_EnergyLvl.eProtection,
    bVal01 := bTWthLowLimit,
    nEn02 := E_BA_EnergyLvl.eEconomy,
    bVal02 := TRUE,
    nEn03 := E_BA_EnergyLvl.eComfort,
    bVal03 := TRUE); // FB_BA_MMUX_B04
Rls(bValuePgm := RlsMMux.bVal); // FB_BA_BV_Op
bRls := Rls.bPresentValue;

METHOD FB_init : BOOL
VAR_INPUT
	bInitRetains : BOOL; // if TRUE, the retain variables are initialized (warm start / cold start)
	bInCopyCode : BOOL;  // if TRUE, the instance afterwards gets moved into the copy code (online change)
END_VAR
OpModMan.iParent		:= THIS^;
OpModMan.iLabel			:= LblCmpHeating.H_OpMod_OpModMan;							
OpModMan.sObjectName	:= '{Idx=01}';								 	 
OpModMan.aStateText[1]	:= txtEvent_Auto;
OpModMan.aStateText[2]	:= txtEvent_Protection;
OpModMan.aStateText[3]	:= txtEvent_Economy;
OpModMan.aStateText[4]	:= txtEvent_Comfort;
OpModMan.nValueRm		:= 1;

OpModPr.iParent			:= THIS^;
OpModPr.iLabel			:= LblCmpHeating.H_OpMod_OpModPr;							
OpModPr.sObjectName		:= '{Idx=01}';								 	 
OpModPr.aStateText[1]	:= txtEvent_Protection; 
OpModPr.aStateText[2]	:= txtEvent_Economy; 
OpModPr.aStateText[3]	:= txtEvent_Comfort; 
OpModPr.nValueRm		:= 1;

Rls.iParent				:= THIS^;
Rls.iLabel				:= LblCmpHeating.H_OpMod_Rls;	
Rls.sObjectName			:= '{Idx=01}';								 	 
Rls.sInactiveText		:= txtEvent_Off;
Rls.sActiveText			:= txtEvent_On;	
Rls.bValueRm			:= FALSE;								
Rls.eToggleMode 		:= E_BA_ToggleMode.eSwitch;	

Sched.iParent											:= THIS^;
Sched.iLabel											:= LblCmpHeating.H_OpMod_Sched;							
Sched.sObjectName										:= '{Idx=01}';								 	 
Sched.aStateText[1]										:= txtEvent_Protection;
Sched.aStateText[2]										:= txtEvent_Economy;
Sched.aStateText[3]										:= txtEvent_Comfort;
Sched.nPredictTime										:= 0;
Sched.nDefaultValue										:= E_BA_EnergyLvl.eProtection;
Sched.bWriteWeekly										:= FALSE;
//	Monday
Sched.aWeek[E_BA_Weekday.eMonday,1].eState				:= E_BA_SchedEntryState.eValue;
Sched.aWeek[E_BA_Weekday.eMonday,1].uValue.udiVal		:= E_BA_EnergyLvl.eComfort;
Sched.aWeek[E_BA_Weekday.eMonday,1].stTime.nHour		:= 6;
Sched.aWeek[E_BA_Weekday.eMonday,1].stTime.nMinute		:= 0;
Sched.aWeek[E_BA_Weekday.eMonday,1].stTime.nSecond		:= 0;
Sched.aWeek[E_BA_Weekday.eMonday,2].eState				:= E_BA_SchedEntryState.eValue;
Sched.aWeek[E_BA_Weekday.eMonday,2].uValue.udiVal		:= E_BA_EnergyLvl.eEconomy;
Sched.aWeek[E_BA_Weekday.eMonday,2].stTime.nHour		:= 20;
Sched.aWeek[E_BA_Weekday.eMonday,2].stTime.nMinute		:= 0;
Sched.aWeek[E_BA_Weekday.eMonday,2].stTime.nSecond		:= 0;
Sched.aWeek[E_BA_Weekday.eMonday,3].eState				:= E_BA_SchedEntryState.eValue;
Sched.aWeek[E_BA_Weekday.eMonday,3].uValue.udiVal		:= E_BA_EnergyLvl.eProtection;
Sched.aWeek[E_BA_Weekday.eMonday,3].stTime.nHour		:= 0;
Sched.aWeek[E_BA_Weekday.eMonday,3].stTime.nMinute		:= 0;
Sched.aWeek[E_BA_Weekday.eMonday,3].stTime.nSecond		:= 0;
//	Tuesday
Sched.aWeek[E_BA_Weekday.eTuesday,1].eState				:= E_BA_SchedEntryState.eValue;
Sched.aWeek[E_BA_Weekday.eTuesday,1].uValue.udiVal		:= E_BA_EnergyLvl.eComfort;
Sched.aWeek[E_BA_Weekday.eTuesday,1].stTime.nHour		:= 6;
Sched.aWeek[E_BA_Weekday.eTuesday,1].stTime.nMinute		:= 0;
Sched.aWeek[E_BA_Weekday.eTuesday,1].stTime.nSecond		:= 0;
Sched.aWeek[E_BA_Weekday.eTuesday,2].eState				:= E_BA_SchedEntryState.eValue;
Sched.aWeek[E_BA_Weekday.eTuesday,2].uValue.udiVal		:= E_BA_EnergyLvl.eEconomy;
Sched.aWeek[E_BA_Weekday.eTuesday,2].stTime.nHour		:= 20;
Sched.aWeek[E_BA_Weekday.eTuesday,2].stTime.nMinute		:= 0;
Sched.aWeek[E_BA_Weekday.eTuesday,2].stTime.nSecond		:= 0;
Sched.aWeek[E_BA_Weekday.eTuesday,3].eState				:= E_BA_SchedEntryState.eValue;
Sched.aWeek[E_BA_Weekday.eTuesday,3].uValue.udiVal		:= E_BA_EnergyLvl.eProtection;
Sched.aWeek[E_BA_Weekday.eTuesday,3].stTime.nHour		:= 0;
Sched.aWeek[E_BA_Weekday.eTuesday,3].stTime.nMinute		:= 0;
Sched.aWeek[E_BA_Weekday.eTuesday,3].stTime.nSecond		:= 0;
//	Wednesday
Sched.aWeek[E_BA_Weekday.eWednesday,1].eState			:= E_BA_SchedEntryState.eValue;
Sched.aWeek[E_BA_Weekday.eWednesday,1].uValue.udiVal	:= E_BA_EnergyLvl.eComfort;
Sched.aWeek[E_BA_Weekday.eWednesday,1].stTime.nHour		:= 6;
Sched.aWeek[E_BA_Weekday.eWednesday,1].stTime.nMinute	:= 0;
Sched.aWeek[E_BA_Weekday.eWednesday,1].stTime.nSecond	:= 0;
Sched.aWeek[E_BA_Weekday.eWednesday,2].eState			:= E_BA_SchedEntryState.eValue;
Sched.aWeek[E_BA_Weekday.eWednesday,2].uValue.udiVal	:= E_BA_EnergyLvl.eEconomy;
Sched.aWeek[E_BA_Weekday.eWednesday,2].stTime.nHour		:= 20;
Sched.aWeek[E_BA_Weekday.eWednesday,2].stTime.nMinute	:= 0;
Sched.aWeek[E_BA_Weekday.eWednesday,2].stTime.nSecond	:= 0;
Sched.aWeek[E_BA_Weekday.eWednesday,3].eState			:= E_BA_SchedEntryState.eValue;
Sched.aWeek[E_BA_Weekday.eWednesday,3].uValue.udiVal	:= E_BA_EnergyLvl.eProtection;
Sched.aWeek[E_BA_Weekday.eWednesday,3].stTime.nHour		:= 0;
Sched.aWeek[E_BA_Weekday.eWednesday,3].stTime.nMinute	:= 0;
Sched.aWeek[E_BA_Weekday.eWednesday,3].stTime.nSecond	:= 0;
//	Thursday
Sched.aWeek[E_BA_Weekday.eThursday,1].eState			:= E_BA_SchedEntryState.eValue;
Sched.aWeek[E_BA_Weekday.eThursday,1].uValue.udiVal		:=E_BA_EnergyLvl.eComfort;
Sched.aWeek[E_BA_Weekday.eThursday,1].stTime.nHour		:= 6;
Sched.aWeek[E_BA_Weekday.eThursday,1].stTime.nMinute	:= 0;
Sched.aWeek[E_BA_Weekday.eThursday,1].stTime.nSecond	:= 0;
Sched.aWeek[E_BA_Weekday.eThursday,2].eState			:= E_BA_SchedEntryState.eValue;
Sched.aWeek[E_BA_Weekday.eThursday,2].uValue.udiVal		:= E_BA_EnergyLvl.eEconomy;
Sched.aWeek[E_BA_Weekday.eThursday,2].stTime.nHour		:= 20;
Sched.aWeek[E_BA_Weekday.eThursday,2].stTime.nMinute	:= 0;
Sched.aWeek[E_BA_Weekday.eThursday,2].stTime.nSecond	:= 0;
Sched.aWeek[E_BA_Weekday.eThursday,3].eState			:= E_BA_SchedEntryState.eValue;
Sched.aWeek[E_BA_Weekday.eThursday,3].uValue.udiVal		:= E_BA_EnergyLvl.eProtection;
Sched.aWeek[E_BA_Weekday.eThursday,3].stTime.nHour		:= 0;
Sched.aWeek[E_BA_Weekday.eThursday,3].stTime.nMinute	:= 0;
Sched.aWeek[E_BA_Weekday.eThursday,3].stTime.nSecond	:= 0;
//	Friday
Sched.aWeek[E_BA_Weekday.eFriday,1].eState				:= E_BA_SchedEntryState.eValue;
Sched.aWeek[E_BA_Weekday.eFriday,1].uValue.udiVal		:= E_BA_EnergyLvl.eComfort;
Sched.aWeek[E_BA_Weekday.eFriday,1].stTime.nHour		:= 6;
Sched.aWeek[E_BA_Weekday.eFriday,1].stTime.nMinute		:= 0;
Sched.aWeek[E_BA_Weekday.eFriday,1].stTime.nSecond		:= 0;
Sched.aWeek[E_BA_Weekday.eFriday,2].eState				:= E_BA_SchedEntryState.eValue;
Sched.aWeek[E_BA_Weekday.eFriday,2].uValue.udiVal		:= E_BA_EnergyLvl.eEconomy;
Sched.aWeek[E_BA_Weekday.eFriday,2].stTime.nHour		:= 20;
Sched.aWeek[E_BA_Weekday.eFriday,2].stTime.nMinute		:= 0;
Sched.aWeek[E_BA_Weekday.eFriday,2].stTime.nSecond		:= 0;
Sched.aWeek[E_BA_Weekday.eFriday,3].eState				:= E_BA_SchedEntryState.eValue;
Sched.aWeek[E_BA_Weekday.eFriday,3].uValue.udiVal		:= E_BA_EnergyLvl.eProtection;
Sched.aWeek[E_BA_Weekday.eFriday,3].stTime.nHour		:= 0;
Sched.aWeek[E_BA_Weekday.eFriday,3].stTime.nMinute		:= 0;
Sched.aWeek[E_BA_Weekday.eFriday,3].stTime.nSecond		:= 0;
END_METHOD

END_FUNCTION_BLOCK

// ---- Templates/POUs/Trade/HeatingSystem/General/FB_BA_HtgLmt.TcPOU
{region '#Template'}
	{attribute 'Version' := '1.0.0.0'}
	{attribute 'Tags' := '"LCID": "1031", "Text": "H, General, HtgCir, Operating mode"'}
	{attribute 'Tags' := '"LCID": "1033", "Text": "H, General, HtgCir, Operating mode"'}
	{attribute 'Description' := '"LCID": "1031", "Text": "Heizgrenzwert"'}
	{attribute 'Description' := '"LCID": "1033", "Text": "Heating limit"'}
{endregion}
FUNCTION_BLOCK FB_BA_HtgLmt EXTENDS FB_BA_View
VAR_INPUT
	fIn						: REAL;
END_VAR
VAR_OUTPUT
	bQ						: BOOL;
END_VAR
VAR_INPUT CONSTANT
	Sp						: FB_BA_AV_Op;	
	Q						: FB_BA_BV_Op;		
END_VAR	
VAR
	Swi2P					: FB_BA_Swi2P;
END_VAR
VAR // added by the converter: edge detectors and wires of the graphical bodies
    _w1 : ANY;
END_VAR

SUPER^(); // FB_BA_View
Sp(); // FB_BA_AV_Op
_w1 := LIMIT(10, Sp.fPresentValue, 32);
Swi2P(bEn := TRUE, fIn := fIn, fOn := _w1, fOff := _w1 + 0.5); // FB_BA_Swi2P
Q(bValuePgm := Swi2P.bQ); // FB_BA_BV_Op
bQ := Q.bPresentValue;

METHOD FB_init : BOOL
VAR_INPUT
	bInitRetains : BOOL; // if TRUE, the retain variables are initialized (warm start / cold start)
	bInCopyCode : BOOL;  // if TRUE, the instance afterwards gets moved into the copy code (online change)
END_VAR
Sp.iParent			:= THIS^;
Sp.iLabel			:= LblCmpHeating.HtgLmt_Sp;
Sp.sObjectName		:= '{Idx=01}';								 	 
Sp.eUnit			:= E_BA_Unit.eTemperature_DegreesCelsius;  
Sp.fValueRm			:= 16.0;
Sp.fCOVIncrement	:= BA2_Param.fDefCOVIncrement;							

Q.iParent			:= THIS^;
Q.iLabel			:= LblCmpHeating.HtgLmt_Q;												 
Q.sObjectName		:= '{Idx=01}';
Q.sActiveText		:= txtEvent_On;
Q.sInactiveText		:= txtEvent_Off;
Q.bValueRm			:= FALSE;								
Q.eToggleMode 		:= E_BA_ToggleMode.eSwitch;
END_METHOD

END_FUNCTION_BLOCK

// ---- Templates/POUs/Universal/Control/PID/FB_BA_PID.TcPOU
{region '#Template'}
	{attribute 'Version' := '1.0.0.0'}
	{attribute 'Tags' := '"LCID": "1031", "Text": "Universal, Control, PID, Loop"'}
	{attribute 'Tags' := '"LCID": "1033", "Text": "Universal, Control, PID, Loop"'}
	{attribute 'Description' := '"LCID": "1031", "Text": "Regler"'}
	{attribute 'Description' := '"LCID": "1033", "Text": "Controller"'}
{endregion}
FUNCTION_BLOCK FB_BA_PID EXTENDS FB_BA_View
VAR_INPUT
	bEn						: BOOL;
	fW						: REAL;
	fX						: REAL;
	bSync					: BOOL;
	fSync					: REAL;
END_VAR
VAR_OUTPUT
	fY						: REAL;
	fMax					: REAL;
	fMin					: REAL;	
END_VAR
VAR_INPUT CONSTANT		 
	Ctrl					: FB_BA_Loop;	
END_VAR

SUPER^(); // FB_BA_View
Ctrl(bEn := bEn, fSetpoint := fW, fCtrlVal := fX, bEnSync := bSync, fValSync := fSync); // FB_BA_Loop
fY := Ctrl.fPresentValue;
fMin := Ctrl.fMinOutputRm;
fMax := Ctrl.fMaxOutputRm;

METHOD FB_init : BOOL
VAR_INPUT
	bInitRetains : BOOL; // if TRUE, the retain variables are initialized (warm start / cold start)
	bInCopyCode : BOOL;  // if TRUE, the instance afterwards gets moved into the copy code (online change)
END_VAR
Ctrl.iParent				:= THIS^;
Ctrl.iLabel					:= LblUniControl.PID_Ctrl; 
Ctrl.sObjectName			:= '{Idx=01}';
Ctrl.eOpMode				:= BA2_Param.nLoop_DefOpMode;								 	 										 
Ctrl.eOutputUnit			:= E_BA_Unit.eOther_Percent;
Ctrl.eActionRm				:= E_BA_Action.eReverse;
Ctrl.fProportionalConstant	:= 3;
Ctrl.fIntegralConstant		:= 180;
Ctrl.fDerivativeConstant	:= 0;
Ctrl.fMaxOutputRm 			:= 100;
Ctrl.fMinOutputRm			:= 0;
Ctrl.fCOVIncrement			:= 0;
Ctrl.nDampConstant			:= 0;
Ctrl.fNeutralZone			:= 0;
END_METHOD

END_FUNCTION_BLOCK

// ---- Templates/POUs/Trade/General/FB_BA_General.TcPOU
{region '#Template'}
	{attribute 'Version' := '1.2.1.0'}
	{attribute 'Tags' := '"LCID": "1031", "Text": "Trade, Plant, General"'}
	{attribute 'Tags' := '"LCID": "1033", "Text": "Trade, Plant, General"'}
	{attribute 'Using' := '"Type": "Template", "URI": "Site"'}
	{attribute 'Description' := '"LCID": "1031", "Text": "Aufruf der Anlagen des Gewerks Allgemein"'}
	{attribute 'Description' := '"LCID": "1033", "Text": "Calling the plants of the trade general"'}
{endregion}
FUNCTION_BLOCK FB_BA_General EXTENDS FB_BA_View
VAR_INPUT
END_VAR
VAR_INPUT CONSTANT
	IFP					: FB_BA_IFP;											 
	EvtGroups			: FB_BA_EvtGroups;											 
	Settings			: FB_BA_Settings;
	Cabinet				: FB_BA_ControlCabinet;				 
	BuildingGlobal		: FB_BA_BuildingGlobal;

	WeatherStation		: FB_BA_RawSubscriber;
	stWeatherStation	: ST_BA_WeatherStation;	
END_VAR

SUPER^(); // FB_BA_View
IFP(); // FB_BA_IFP
Settings(fTWth := stWeatherStation.fOutsideTemperature); // FB_BA_Settings
EvtGroups(); // FB_BA_EvtGroups
Cabinet(); // FB_BA_ControlCabinet
BuildingGlobal(); // FB_BA_BuildingGlobal
WeatherStation(xData := stWeatherStation); // FB_BA_RawSubscriber

METHOD FB_init : BOOL
VAR_INPUT
	bInitRetains : BOOL; // if TRUE, the retain variables are initialized (warm start / cold start)
	bInCopyCode : BOOL;  // if TRUE, the instance afterwards gets moved into the copy code (online change)
END_VAR
IFP.iParent						:= THIS^;	
IFP.sObjectName					:= '{ISP01}';
IFP.sDescription				:= '{Information focal point}';
IFP.eDPADMode					:= E_BA_DPADMode.eInclude;		

EvtGroups.iParent				:= THIS^;	
EvtGroups.sObjectName			:= '{EVG01}';
EvtGroups.sDescription			:= '{Event groups}';
EvtGroups.eDPADMode				:= E_BA_DPADMode.eInclude;									

Settings.iParent				:= THIS^;										 
Settings.sObjectName			:= '{SYP01}';
Settings.sDescription			:= '{System parameters}';
Settings.eDPADMode				:= E_BA_DPADMode.eInclude;

Cabinet.iParent					:= THIS^;	
Cabinet.sObjectName				:= '{CCB01}';
Cabinet.sDescription			:= '{Control cabinet}';									 
Cabinet.eDPADMode				:= E_BA_DPADMode.eInclude;
				 
BuildingGlobal.iParent			:= THIS^;	
BuildingGlobal.sObjectName		:= '{GBD01}';														 
BuildingGlobal.sDescription		:= '{global building Data}';														 
BuildingGlobal.eDPADMode		:= E_BA_DPADMode.eInclude;

WeatherStation.Subject			:= Site.WeatherStation_Subject;
WeatherStation.sTarget			:= Site.WeatherStation_NetId;
END_METHOD

END_FUNCTION_BLOCK

// ---- Templates/POUs/Trade/General/IFP/FB_BA_IFP.TcPOU
{region '#Template'}
	{attribute 'Version' := '1.2.1.0'}
	{attribute 'Tags' := '"LCID": "1031", "Text": "General, Settings, Project, Basics"'}
	{attribute 'Tags' := '"LCID": "1033", "Text": "General, Settings, Project, Basics"'}
	{attribute 'Description' := '"LCID": "1031", "Text": "Basis Einstellungen der Steuerung, system services"'}
	{attribute 'Description' := '"LCID": "1033", "Text": "Basic settings of the control"'}
{endregion}
FUNCTION_BLOCK FB_BA_IFP EXTENDS FB_BA_View
VAR_INPUT
END_VAR
VAR_INPUT CONSTANT
	Trend				: FB_BA_TrendLogging;	
	Project				: FB_BA_ProjectEx;
END_VAR
VAR_OUTPUT
END_VAR
VAR
	LblProject			: FB_BA_Label2x :=(iAggregate:=LblAggregates_AutomationStationEquipment,	 iFunction:=LblControl_BACnetDevice);
END_VAR

SUPER^(); // FB_BA_View
Trend(); // FB_BA_TrendLogging
// connect a UPS-monitoring FB at this input
Project(); // FB_BA_ProjectEx

METHOD FB_init : BOOL
VAR_INPUT
	bInitRetains : BOOL; // if TRUE, the retain variables are initialized (warm start / cold start)
	bInCopyCode : BOOL;  // if TRUE, the instance afterwards gets moved into the copy code (online change)
END_VAR
Project.iParent						:= THIS^;
Project.iLabel						:= LblProject;

Project.tPrsData_DefaultPeriod 		:= T#30M;
Project.tPrsData_ComissioningPeriod := T#10M;

Trend.iParent						:= THIS^;
Trend.iLabel						:= LblControl_TrendLogging;
Trend.sObjectName					:= '{Idx=01}';
Trend.eDPADMode						:= E_BA_DPADMode.eInclude;
END_METHOD

END_FUNCTION_BLOCK

// ---- Templates/POUs/Universal/Control/Trend/FB_BA_TrendLogging.TcPOU
{region '#Template'}
	{attribute 'Version' := '1.2.1.0'}
	{attribute 'Tags' := '"LCID": "1031", "Text": "Universal, Control, Trend"'}
	{attribute 'Tags' := '"LCID": "1033", "Text": "Universal, Control, Trend"'}
	{attribute 'Using' := '"Type": "Template", "URI": "EC_AMEV"'}
	{attribute 'Using' := '"Type": "Template", "URI": "BA2_Param"'}
	{attribute 'Description' := '"LCID": "1031", "Text": "Trend"'}
	{attribute 'Description' := '"LCID": "1033", "Text": "Trend"'}
{endregion}			 
FUNCTION_BLOCK FB_BA_TrendLogging EXTENDS FB_BA_View
VAR_INPUT
END_VAR
VAR_OUTPUT
END_VAR
VAR_INPUT CONSTANT
	Trends						: ARRAY[1..TREND_COUNT] OF FB_BA_Trend;								
END_VAR
VAR
	i							: UDINT;
END_VAR
VAR CONSTANT
	TREND_COUNT						: UDINT := 30;
END_VAR

SUPER^();

FOR i := 1 TO TREND_COUNT DO
	Trends[i]();
END_FOR

METHOD FB_init : BOOL
VAR_INPUT
	bInitRetains : BOOL; // if TRUE, the retain variables are initialized (warm start / cold start)
	bInCopyCode : BOOL;  // if TRUE, the instance afterwards gets moved into the copy code (online change)
END_VAR 
VAR
	sIdx	: STRING;
END_VAR
FOR i := 1 TO TREND_COUNT DO
	sIdx := CONCAT(TO_STRING(i),'}');;

	Trends[i].iParent					:= THIS^;
	Trends[i].iLabel					:= LblFunctions_ObjectTrendLog;
	Trends[i].sObjectName				:= CONCAT('{Idx=',sIdx);
	Trends[i].bEnable					:= BA2_Param.bTrend_DefLogEnable;
	Trends[i].stStartTime				:= BA2_Param.stTrend_DefStartTime;
	Trends[i].stStopTime				:= BA2_Param.stTrend_DefStopTime;	
	Trends[i].nLogInterval 				:= BA2_Param.nTrend_DefLogInterval;
	Trends[i].bStopOnFull				:= BA2_Param.bTrend_DefStopOnFull;
	Trends[i].nBufferSize 				:= BA2_Param.nTrend_BufferSize;
	Trends[i].eLoggingType				:= BA2_Param.eTrend_DefLoggingType;	
	Trends[i].nEventClassID				:= EC_ID.NC80;
	Trends[i].nNotificationThreshold	:= BA2_Param.nTrend_DefNotificationThreshold;
	Trends[i].aEventTransitionText[1]	:= txtEvent_Offnormal;
	Trends[i].aEventTransitionText[2]	:= txtEvent_None;
	Trends[i].aEventTransitionText[3]	:= txtEvent_Normal;
	Trends[i].bEventDetectionEnable		:= FALSE;
	Trends[i].aEventEnable[1]			:= TRUE;			//	to_offnormal
	Trends[i].aEventEnable[2]			:= TRUE;			//	to_fault
	Trends[i].aEventEnable[3]			:= TRUE;			//	to_normal	
	Trends[i].bAcknowledgeRm			:= FALSE;		
END_FOR
END_METHOD

END_FUNCTION_BLOCK

// ---- Templates/POUs/Trade/General/IFP/Project/FB_BA_ProjectEx.TcPOU
{region '#Template'}
	{attribute 'Version' := '1.2.1.0'}
	{attribute 'Tags' := '"LCID": "1031", "Text": "General, Settings, Project, Basics"'}
	{attribute 'Tags' := '"LCID": "1033", "Text": "General, Settings, Project, Basics"'}
	{attribute 'Description' := '"LCID": "1031", "Text": "Projektspezifische Informationen"'}
	{attribute 'Description' := '"LCID": "1033", "Text": "Project specific informations"'}
{endregion}
FUNCTION_BLOCK FB_BA_ProjectEx EXTENDS FB_BA_Project
VAR_INPUT CONSTANT PERSISTENT
	{attribute 'parameterCategory' := 'Persistent Data'}
	tPrsData_DefaultPeriod : TIME := T#30M;
	{attribute 'parameterCategory' := 'Persistent Data'}
	tPrsData_ComissioningPeriod : TIME := T#10M;
END_VAR
VAR_INPUT CONSTANT
	{attribute 'parameterCategory' := 'Persistent Data'}
	bPrsData_ManualWriteData : BOOL;
END_VAR
VAR_INPUT
	bWrtPrsOnPowerFail		: BOOL;
END_VAR
VAR_OUTPUT
	nPrsDataWritten			: UINT;
END_VAR

SUPER^();

OnInitCycle();
PersistentData();

METHOD PROTECTED OnInitCycle
VAR
	_stVersion		: ST_LibVersion;
END_VAR
VAR CONSTANT
	FORMAT			: STRING		:= '%d.%d.%d.%d';
END_VAR
CASE (State) OF
	E_BA_ObjectState.eInstanceInit1:
		// Refresh runtime information:
		{IF defined (pou: F_GetVersion)}
			_stVersion := F_GetVersion();
			
			BA_Globals.Format(
				pFormatString := ADR(FORMAT),
				arg1:=F_UINT(_stVersion.iMajor),
				arg2:=F_UINT(_stVersion.iMinor),
				arg3:=F_UINT(_stVersion.iBuild),
				arg4:=F_UINT(_stVersion.iRevision),
			
				pDstString := ADR(stVersion.Project),
				nDstSize := SIZEOF(stVersion.Project)
			);
		{END_IF}
		
END_CASE
END_METHOD

METHOD PROTECTED PersistentData
VAR_INST
	nOnlineChangeCnt		:	UDINT;
	iStep					:	INT;
	fbTon					:	TON;
	fbResetOnlineChange		:	TON;
	rtigManual				:	R_TRIG;
	trigUPS					:	R_TRIG;
	rFinishTrig				:	R_TRIG;
	WrtPersistDat			:	FB_BA_WrtPersistDat;
END_VAR
VAR CONSTANT
	DETECT_COMISSIONING_DURATION : TIME := T#60M;
END_VAR
IF	TwinCAT_SystemInfoVarList._AppInfo.OnlineChangeCnt <> nOnlineChangeCnt THEN
	nOnlineChangeCnt := TwinCAT_SystemInfoVarList._AppInfo.OnlineChangeCnt;
	fbResetOnlineChange(IN := FALSE);
	fbTon(IN := FALSE);
	iStep := 10;
END_IF

IF	tPrsData_DefaultPeriod < T#600S THEN
	tPrsData_DefaultPeriod	:= T#1800S;
END_IF

IF	tPrsData_ComissioningPeriod < T#30S THEN
	tPrsData_ComissioningPeriod	:= T#300S;
END_IF

CASE	iStep	OF
	0:
		fbTon(IN := NOT fbTon.Q,PT := tPrsData_DefaultPeriod);
	10:
		fbTon(IN := NOT fbTon.Q,PT := tPrsData_ComissioningPeriod);
		fbResetOnlineChange(IN := TRUE, PT := DETECT_COMISSIONING_DURATION);
		
		IF	fbResetOnlineChange.Q THEN
			iStep := 0;
			fbResetOnlineChange(IN := FALSE);
		END_IF
END_CASE
 
rtigManual(CLK := bPrsData_ManualWriteData);
bPrsData_ManualWriteData := FALSE;

trigUPS(CLK := bWrtPrsOnPowerFail);

// Write persistent data:
WrtPersistDat(bStt:=(fbTon.Q OR rtigManual.Q OR trigUPS.Q));
rFinishTrig(CLK:=(WrtPersistDat.bBusy AND NOT WrtPersistDat.bErr));

IF (rFinishTrig.Q) THEN
	nPrsDataWritten := (nPrsDataWritten+1);
END_IF
END_METHOD

END_FUNCTION_BLOCK

// ---- Templates/POUs/Trade/General/EventClasses/FB_BA_EvtGroups.TcPOU
{region '#Template'}
	{attribute 'Version' := '1.2.2.0'}
	{attribute 'Tags' := '"LCID": "1031", "Text": "General, Cabinet, Control cabinet, Event groups, Categories, Notification classes, Event classes"'}
	{attribute 'Tags' := '"LCID": "1033", "Text": "General, Cabinet, Control cabinet, Event groups, Categories, Notification classes, Event classes"'}
	{attribute 'Using' := '"Type": "Template", "URI": "EC_AMEV"'}
	{attribute 'Description' := '"LCID": "1031", "Text": "Ereignisgruppen, Kategorien"'}
	{attribute 'Description' := '"LCID": "1033", "Text": "Event groups, categories"'}
{endregion}
FUNCTION_BLOCK FB_BA_EvtGroups EXTENDS FB_BA_View
VAR_INPUT CONSTANT
	LifeSafety						: FB_BA_EvtCategory;
	SafetyMsg						: FB_BA_EvtCategory;
	AlarmMsg						: FB_BA_EvtCategory;
	FaultMsg						: FB_BA_EvtCategory;
	MaintenanceMsg01				: FB_BA_EvtCategory;
	MaintenanceMsg02				: FB_BA_EvtCategory;
	SystemMsg						: FB_BA_EvtCategory;
	ManualOp						: FB_BA_EvtCategory;
	OtherMsg						: FB_BA_EvtCategory;
END_VAR

SUPER^(); // FB_BA_View
LifeSafety(); // FB_BA_EvtCategory
SafetyMsg(); // FB_BA_EvtCategory
AlarmMsg(); // FB_BA_EvtCategory
FaultMsg(); // FB_BA_EvtCategory
MaintenanceMsg01(); // FB_BA_EvtCategory
MaintenanceMsg02(); // FB_BA_EvtCategory
SystemMsg(); // FB_BA_EvtCategory
ManualOp(); // FB_BA_EvtCategory
OtherMsg(); // FB_BA_EvtCategory

METHOD FB_init : BOOL
VAR_INPUT
	bInitRetains : BOOL; // if TRUE, the retain variables are initialized (warm start / cold start)
	bInCopyCode : BOOL;  // if TRUE, the instance afterwards gets moved into the copy code (online change)
END_VAR
//===================================================================
// Ereigniskategorie - Gefahr für Leben // Event category - Danger to life
// Brandalarm, Überfall // Fire alarm, robbery
LifeSafety.iParent							:= THIS^;
LifeSafety.iLabel							:= LblControl_EvtCategoryLifeSafty;									  
LifeSafety.sObjectName						:= '{Idx=01}';
LifeSafety.eDPADMode						:= E_BA_DPADMode.eInclude;																						
LifeSafety.EC.nInstanceID						:= EC_ID.NC10;
LifeSafety.EC.sObjectName						:= '{Idx=10}';
LifeSafety.EC.eEventType						:= E_BA_EventType.eAlarm;
LifeSafety.EC.aPriority[1]						:= 10;
LifeSafety.EC.aPriority[2]						:= 11;
LifeSafety.EC.aPriority[3]						:= 12;
LifeSafety.EC.eAlarmMode						:= E_BA_AlarmMode.eExtended;	//Erweiterter Alarm
//===================================================================		
// Ereigniskategorie - Gefahrenmeldung, Sicherheitsmeldung // Event category - hazard alert, safety message
// Einbruch, unberechtigter Zutritt // Burglary, unauthorised entry
SafetyMsg.iParent							:= THIS^;
SafetyMsg.iLabel							:= LblControl_EvtCategorySaftyMessage;									  
SafetyMsg.sObjectName						:= '{Idx=01}';
SafetyMsg.eDPADMode							:= E_BA_DPADMode.eInclude;																						
SafetyMsg.EC.nInstanceID						:= EC_ID.NC20;
SafetyMsg.EC.sObjectName						:= '{Idx=20}';
SafetyMsg.EC.eEventType							:= E_BA_EventType.eAlarm;
SafetyMsg.EC.aPriority[1]						:= 40;
SafetyMsg.EC.aPriority[2]						:= 41;
SafetyMsg.EC.aPriority[3]						:= 42;
SafetyMsg.EC.eAlarmMode						:= E_BA_AlarmMode.eExtended;	//Erweiterter Alarm

